FONT_5X12:ARRAY[0..255,0..9]OF BYTE :=[
16#00,16#00,16#00,16#00,16#00,16#00,16#00,16#00,16#00,16#00,	// 16#00
16#FE,16#01,16#49,16#02,16#81,16#02,16#49,16#02,16#FE,16#01,	// 16#01
16#FE,16#01,16#B7,16#03,16#7F,16#03,16#B7,16#03,16#FE,16#01,	// 16#02
16#7C,16#00,16#FE,16#01,16#F8,16#07,16#FE,16#01,16#7C,16#00,	// 16#03
16#70,16#00,16#FC,16#01,16#FF,16#07,16#FC,16#01,16#70,16#00,	// 16#04
16#60,16#00,16#EE,16#02,16#FF,16#03,16#EE,16#02,16#60,16#00,	// 16#05
16#70,16#00,16#FC,16#02,16#FF,16#03,16#FC,16#02,16#70,16#00,	// 16#06
16#00,16#00,16#00,16#00,16#00,16#00,16#00,16#00,16#00,16#00,	// 16#07
16#00,16#00,16#00,16#00,16#00,16#00,16#00,16#00,16#00,16#00,	// 16#08
16#00,16#00,16#00,16#00,16#00,16#00,16#00,16#00,16#00,16#00,	// 16#09
16#00,16#00,16#00,16#00,16#00,16#00,16#00,16#00,16#00,16#00,	// 16#0A
16#C0,16#01,16#20,16#02,16#34,16#02,16#CC,16#01,16#1C,16#00,	// 16#0B
16#1C,16#01,16#E2,16#03,16#22,16#01,16#1C,16#00,16#00,16#00,	// 16#0C
16#00,16#00,16#00,16#00,16#00,16#00,16#00,16#00,16#00,16#00,	// 16#0D
16#00,16#03,16#FE,16#03,16#C5,16#00,16#FF,16#00,16#00,16#00,	// 16#0E
16#50,16#01,16#A0,16#00,16#B0,16#01,16#A0,16#00,16#50,16#01,	// 16#0F
16#FC,16#01,16#F8,16#00,16#70,16#00,16#20,16#00,16#00,16#00,	// 16#10
16#20,16#00,16#70,16#00,16#F8,16#00,16#FC,16#01,16#00,16#00,	// 16#11
16#88,16#00,16#04,16#01,16#FE,16#03,16#04,16#01,16#88,16#00,	// 16#12
16#00,16#00,16#7C,16#03,16#00,16#00,16#7C,16#03,16#00,16#00,	// 16#13
16#3C,16#00,16#FE,16#03,16#02,16#00,16#FE,16#03,16#00,16#00,	// 16#14
16#2C,16#01,16#52,16#02,16#52,16#02,16#A4,16#01,16#00,16#00,	// 16#15
16#00,16#03,16#00,16#03,16#00,16#03,16#00,16#03,16#00,16#00,	// 16#16
16#88,16#04,16#04,16#05,16#FE,16#07,16#04,16#05,16#88,16#04,	// 16#17
16#08,16#00,16#04,16#00,16#FE,16#03,16#04,16#00,16#08,16#00,	// 16#18
16#80,16#00,16#00,16#01,16#FC,16#03,16#00,16#01,16#80,16#00,	// 16#19
16#20,16#00,16#A8,16#00,16#70,16#00,16#20,16#00,16#00,16#00,	// 16#1A
16#20,16#00,16#70,16#00,16#A8,16#00,16#20,16#00,16#00,16#00,	// 16#1B
16#E0,16#00,16#80,16#00,16#80,16#00,16#80,16#00,16#00,16#00,	// 16#1C
16#20,16#00,16#F8,16#00,16#20,16#00,16#F8,16#00,16#20,16#00,	// 16#1D
16#80,16#00,16#E0,16#00,16#F8,16#00,16#E0,16#00,16#80,16#00,	// 16#1E
16#08,16#00,16#38,16#00,16#F8,16#00,16#38,16#00,16#08,16#00,	// 16#1F
16#00,16#00,16#00,16#00,16#00,16#00,16#00,16#00,16#00,16#00,	// 16#20
16#00,16#00,16#00,16#00,16#7E,16#03,16#00,16#00,16#00,16#00,	// 16#21
16#00,16#00,16#0F,16#00,16#00,16#00,16#0F,16#00,16#00,16#00,	// 16#22
16#48,16#00,16#FE,16#01,16#48,16#00,16#FE,16#01,16#48,16#00,	// 16#23
16#18,16#01,16#26,16#02,16#44,16#06,16#88,16#01,16#00,16#00,	// 16#24
16#06,16#03,16#E6,16#00,16#18,16#03,16#06,16#03,16#00,16#00,	// 16#25
16#DC,16#01,16#22,16#02,16#5C,16#02,16#80,16#01,16#40,16#02,	// 16#26
16#00,16#00,16#00,16#00,16#0B,16#00,16#07,16#00,16#00,16#00,	// 16#27
16#00,16#00,16#FC,16#01,16#02,16#02,16#00,16#00,16#00,16#00,	// 16#28
16#00,16#00,16#02,16#02,16#FC,16#01,16#00,16#00,16#00,16#00,	// 16#29
16#48,16#00,16#30,16#00,16#FC,16#00,16#30,16#00,16#48,16#00,	// 16#2A
16#20,16#00,16#20,16#00,16#F8,16#00,16#20,16#00,16#20,16#00,	// 16#2B
16#00,16#00,16#00,16#0B,16#00,16#07,16#00,16#00,16#00,16#00,	// 16#2C
16#20,16#00,16#20,16#00,16#20,16#00,16#20,16#00,16#00,16#00,	// 16#2D
16#00,16#00,16#00,16#03,16#00,16#03,16#00,16#00,16#00,16#00,	// 16#2E
16#00,16#03,16#E0,16#00,16#18,16#00,16#06,16#00,16#00,16#00,	// 16#2F
16#FC,16#03,16#02,16#02,16#02,16#02,16#FE,16#01,16#00,16#00,	// 16#30
16#08,16#02,16#04,16#02,16#FE,16#03,16#00,16#02,16#00,16#00,	// 16#31
16#8C,16#03,16#42,16#02,16#22,16#02,16#1C,16#02,16#00,16#00,	// 16#32
16#04,16#01,16#22,16#02,16#22,16#02,16#DC,16#01,16#00,16#00,	// 16#33
16#60,16#00,16#58,16#00,16#44,16#00,16#FE,16#03,16#00,16#00,	// 16#34
16#3E,16#01,16#22,16#02,16#22,16#02,16#C2,16#01,16#00,16#00,	// 16#35
16#F8,16#01,16#14,16#02,16#12,16#02,16#E2,16#01,16#00,16#00,	// 16#36
16#02,16#00,16#82,16#03,16#62,16#00,16#1E,16#00,16#00,16#00,	// 16#37
16#DC,16#01,16#22,16#02,16#22,16#02,16#DC,16#01,16#00,16#00,	// 16#38
16#3C,16#02,16#42,16#02,16#42,16#01,16#FC,16#00,16#00,16#00,	// 16#39
16#00,16#00,16#30,16#03,16#30,16#03,16#00,16#00,16#00,16#00,	// 16#3A
16#00,16#00,16#30,16#0B,16#30,16#07,16#00,16#00,16#00,16#00,	// 16#3B
16#60,16#00,16#90,16#00,16#08,16#01,16#04,16#02,16#00,16#00,	// 16#3C
16#A0,16#00,16#A0,16#00,16#A0,16#00,16#A0,16#00,16#00,16#00,	// 16#3D
16#04,16#02,16#08,16#01,16#90,16#00,16#60,16#00,16#00,16#00,	// 16#3E
16#0C,16#00,16#02,16#00,16#62,16#03,16#1C,16#00,16#00,16#00,	// 16#3F
16#FC,16#01,16#02,16#02,16#62,16#02,16#7C,16#02,16#00,16#00,	// 16#40
16#FC,16#03,16#22,16#00,16#22,16#00,16#FC,16#03,16#00,16#00,	// 16#41
16#FE,16#03,16#22,16#02,16#22,16#02,16#DC,16#01,16#00,16#00,	// 16#42
16#FC,16#01,16#02,16#02,16#02,16#02,16#0C,16#01,16#00,16#00,	// 16#43
16#FE,16#03,16#02,16#02,16#02,16#02,16#FC,16#01,16#00,16#00,	// 16#44
16#FE,16#03,16#22,16#02,16#22,16#02,16#22,16#02,16#00,16#00,	// 16#45
16#FE,16#03,16#22,16#00,16#22,16#00,16#22,16#00,16#00,16#00,	// 16#46
16#FC,16#01,16#02,16#02,16#42,16#02,16#CC,16#01,16#00,16#00,	// 16#47
16#FE,16#03,16#20,16#00,16#20,16#00,16#FE,16#03,16#00,16#00,	// 16#48
16#00,16#00,16#02,16#02,16#FE,16#03,16#02,16#02,16#00,16#00,	// 16#49
16#80,16#01,16#02,16#02,16#FE,16#01,16#02,16#00,16#00,16#00,	// 16#4A
16#FE,16#03,16#20,16#00,16#D8,16#00,16#06,16#03,16#00,16#00,	// 16#4B
16#FE,16#03,16#00,16#02,16#00,16#02,16#00,16#02,16#00,16#00,	// 16#4C
16#FE,16#03,16#18,16#00,16#18,16#00,16#FE,16#03,16#00,16#00,	// 16#4D
16#FE,16#03,16#18,16#00,16#60,16#00,16#FE,16#03,16#00,16#00,	// 16#4E
16#FC,16#01,16#02,16#02,16#02,16#02,16#FC,16#01,16#00,16#00,	// 16#4F
16#FE,16#03,16#22,16#00,16#22,16#00,16#1C,16#00,16#00,16#00,	// 16#50
16#FC,16#01,16#02,16#02,16#02,16#06,16#FC,16#09,16#00,16#00,	// 16#51
16#FE,16#03,16#62,16#00,16#A2,16#00,16#1C,16#03,16#00,16#00,	// 16#52
16#9C,16#01,16#22,16#02,16#22,16#02,16#CC,16#01,16#00,16#00,	// 16#53
16#02,16#00,16#02,16#00,16#FE,16#03,16#02,16#00,16#02,16#00,	// 16#54
16#FE,16#01,16#00,16#02,16#00,16#02,16#FE,16#01,16#00,16#00,	// 16#55
16#3E,16#00,16#C0,16#00,16#00,16#03,16#FE,16#00,16#00,16#00,	// 16#56
16#FE,16#03,16#80,16#00,16#80,16#00,16#FE,16#03,16#00,16#00,	// 16#57
16#8E,16#03,16#70,16#00,16#70,16#00,16#8E,16#03,16#00,16#00,	// 16#58
16#0E,16#00,16#30,16#00,16#C0,16#03,16#30,16#00,16#0E,16#00,	// 16#59
16#82,16#03,16#62,16#02,16#1A,16#02,16#06,16#02,16#00,16#00,	// 16#5A
16#00,16#00,16#FE,16#03,16#02,16#02,16#00,16#00,16#00,16#00,	// 16#5B
16#06,16#00,16#18,16#00,16#E0,16#00,16#00,16#03,16#00,16#00,	// 16#5C
16#00,16#00,16#02,16#02,16#FE,16#03,16#00,16#00,16#00,16#00,	// 16#5D
16#00,16#00,16#04,16#00,16#02,16#00,16#04,16#00,16#00,16#00,	// 16#5E
16#00,16#08,16#00,16#08,16#00,16#08,16#00,16#08,16#00,16#08,	// 16#5F
16#00,16#00,16#07,16#00,16#0B,16#00,16#00,16#00,16#00,16#00,	// 16#60
16#80,16#01,16#50,16#02,16#50,16#02,16#E0,16#03,16#00,16#00,	// 16#61
16#FE,16#03,16#10,16#02,16#10,16#02,16#E0,16#01,16#00,16#00,	// 16#62
16#E0,16#01,16#10,16#02,16#10,16#02,16#10,16#02,16#00,16#00,	// 16#63
16#E0,16#01,16#10,16#02,16#10,16#02,16#FE,16#03,16#00,16#00,	// 16#64
16#E0,16#01,16#90,16#02,16#90,16#02,16#E0,16#02,16#00,16#00,	// 16#65
16#10,16#00,16#FC,16#03,16#12,16#00,16#00,16#00,16#00,16#00,	// 16#66
16#E0,16#01,16#10,16#0A,16#10,16#0A,16#F0,16#07,16#00,16#00,	// 16#67
16#FE,16#03,16#10,16#00,16#10,16#00,16#E0,16#03,16#00,16#00,	// 16#68
16#00,16#00,16#00,16#02,16#F4,16#03,16#00,16#02,16#00,16#00,	// 16#69
16#00,16#04,16#00,16#08,16#F4,16#07,16#00,16#00,16#00,16#00,	// 16#6A
16#FE,16#03,16#C0,16#00,16#20,16#01,16#10,16#02,16#00,16#00,	// 16#6B
16#00,16#00,16#02,16#02,16#FE,16#03,16#00,16#02,16#00,16#00,	// 16#6C
16#F0,16#03,16#20,16#00,16#20,16#00,16#F0,16#03,16#00,16#00,	// 16#6D
16#F0,16#03,16#20,16#00,16#10,16#00,16#E0,16#03,16#00,16#00,	// 16#6E
16#E0,16#01,16#10,16#02,16#10,16#02,16#E0,16#01,16#00,16#00,	// 16#6F
16#F0,16#0F,16#10,16#02,16#10,16#02,16#E0,16#01,16#00,16#00,	// 16#70
16#E0,16#01,16#10,16#02,16#10,16#02,16#F0,16#0F,16#00,16#00,	// 16#71
16#10,16#00,16#E0,16#03,16#10,16#00,16#30,16#00,16#00,16#00,	// 16#72
16#20,16#01,16#50,16#02,16#90,16#02,16#20,16#01,16#00,16#00,	// 16#73
16#10,16#00,16#FC,16#03,16#10,16#02,16#00,16#00,16#00,16#00,	// 16#74
16#F0,16#01,16#00,16#02,16#00,16#02,16#F0,16#03,16#00,16#00,	// 16#75
16#30,16#00,16#C0,16#00,16#00,16#03,16#F0,16#00,16#00,16#00,	// 16#76
16#F0,16#03,16#00,16#01,16#00,16#01,16#F0,16#03,16#00,16#00,	// 16#77
16#30,16#03,16#C0,16#00,16#C0,16#00,16#30,16#03,16#00,16#00,	// 16#78
16#F0,16#09,16#00,16#0A,16#00,16#0A,16#F0,16#07,16#00,16#00,	// 16#79
16#10,16#03,16#90,16#02,16#50,16#02,16#30,16#02,16#00,16#00,	// 16#7A
16#20,16#00,16#DC,16#01,16#02,16#02,16#00,16#00,16#00,16#00,	// 16#7B
16#00,16#00,16#00,16#00,16#EF,16#03,16#00,16#00,16#00,16#00,	// 16#7C
16#00,16#00,16#02,16#02,16#DC,16#01,16#20,16#00,16#00,16#00,	// 16#7D
16#04,16#00,16#02,16#00,16#04,16#00,16#02,16#00,16#00,16#00,	// 16#7E
16#E0,16#03,16#18,16#02,16#06,16#02,16#18,16#02,16#E0,16#03,	// 16#7F
16#FC,16#01,16#02,16#0A,16#02,16#06,16#0C,16#01,16#00,16#00,	// 16#80
16#F0,16#01,16#06,16#02,16#00,16#02,16#F6,16#03,16#00,16#00,	// 16#81
16#E0,16#01,16#94,16#02,16#92,16#02,16#E2,16#02,16#00,16#00,	// 16#82
16#24,16#01,16#92,16#02,16#92,16#02,16#E4,16#03,16#00,16#00,	// 16#83
16#20,16#01,16#96,16#02,16#90,16#02,16#E6,16#03,16#00,16#00,	// 16#84
16#22,16#01,16#92,16#02,16#94,16#02,16#E0,16#03,16#00,16#00,	// 16#85
16#20,16#01,16#94,16#02,16#9A,16#02,16#E4,16#03,16#00,16#00,	// 16#86
16#E0,16#09,16#10,16#0A,16#10,16#06,16#10,16#02,16#00,16#00,	// 16#87
16#E4,16#01,16#92,16#02,16#92,16#02,16#E4,16#02,16#00,16#00,	// 16#88
16#E0,16#01,16#96,16#02,16#90,16#02,16#E6,16#02,16#00,16#00,	// 16#89
16#E2,16#01,16#92,16#02,16#94,16#02,16#E0,16#02,16#00,16#00,	// 16#8A
16#00,16#00,16#16,16#02,16#F0,16#03,16#06,16#02,16#00,16#00,	// 16#8B
16#04,16#00,16#12,16#02,16#F2,16#03,16#04,16#02,16#00,16#00,	// 16#8C
16#00,16#00,16#12,16#02,16#F2,16#03,16#04,16#02,16#00,16#00,	// 16#8D
16#F8,16#03,16#45,16#00,16#44,16#00,16#F9,16#03,16#00,16#00,	// 16#8E
16#F0,16#03,16#4A,16#00,16#4D,16#00,16#F2,16#03,16#00,16#00,	// 16#8F
16#F8,16#03,16#4A,16#02,16#49,16#02,16#49,16#02,16#00,16#00,	// 16#90
16#00,16#01,16#90,16#02,16#F0,16#01,16#90,16#02,16#60,16#00,	// 16#91
16#F8,16#03,16#4C,16#00,16#FC,16#03,16#44,16#02,16#00,16#00,	// 16#92
16#E4,16#01,16#12,16#02,16#12,16#02,16#E4,16#01,16#00,16#00,	// 16#93
16#E0,16#01,16#16,16#02,16#10,16#02,16#E6,16#01,16#00,16#00,	// 16#94
16#E0,16#01,16#12,16#02,16#12,16#02,16#E4,16#01,16#00,16#00,	// 16#95
16#F4,16#01,16#02,16#02,16#02,16#02,16#F4,16#03,16#00,16#00,	// 16#96
16#F2,16#01,16#02,16#02,16#04,16#02,16#F0,16#03,16#00,16#00,	// 16#97
16#F0,16#09,16#06,16#0A,16#00,16#0A,16#F6,16#07,16#00,16#00,	// 16#98
16#F8,16#01,16#05,16#02,16#04,16#02,16#F9,16#01,16#00,16#00,	// 16#99
16#FC,16#01,16#01,16#02,16#00,16#02,16#FD,16#03,16#00,16#00,	// 16#9A
16#E0,16#03,16#90,16#01,16#70,16#01,16#F8,16#00,16#00,16#00,	// 16#9B
16#20,16#03,16#FC,16#03,16#22,16#02,16#04,16#03,16#00,16#00,	// 16#9C
16#FE,16#03,16#E1,16#03,16#1D,16#02,16#FF,16#01,16#00,16#00,	// 16#9D
16#88,16#00,16#50,16#00,16#20,16#00,16#50,16#00,16#88,16#00,	// 16#9E
16#00,16#04,16#20,16#08,16#FE,16#07,16#21,16#00,16#00,16#00,	// 16#9F
16#20,16#01,16#94,16#02,16#92,16#02,16#E2,16#03,16#00,16#00,	// 16#A0
16#00,16#00,16#14,16#02,16#F2,16#03,16#02,16#02,16#00,16#00,	// 16#A1
16#E0,16#01,16#14,16#02,16#12,16#02,16#E2,16#01,16#00,16#00,	// 16#A2
16#F0,16#01,16#04,16#02,16#02,16#02,16#F2,16#03,16#00,16#00,	// 16#A3
16#F4,16#03,16#22,16#00,16#14,16#00,16#E2,16#03,16#00,16#00,	// 16#A4
16#FA,16#03,16#31,16#00,16#62,16#00,16#F9,16#03,16#00,16#00,	// 16#A5
16#90,16#00,16#AA,16#00,16#AA,16#00,16#BC,16#00,16#00,16#00,	// 16#A6
16#9C,16#00,16#A2,16#00,16#A2,16#00,16#9C,16#00,16#00,16#00,	// 16#A7
16#C0,16#01,16#36,16#02,16#00,16#02,16#00,16#01,16#00,16#00,	// 16#A8
16#F8,16#01,16#F4,16#02,16#54,16#02,16#A4,16#02,16#F8,16#01,	// 16#A9
16#40,16#00,16#40,16#00,16#40,16#00,16#C0,16#01,16#00,16#00,	// 16#AA
16#80,16#01,16#6E,16#00,16#50,16#03,16#CC,16#02,16#00,16#00,	// 16#AB
16#80,16#01,16#6E,16#00,16#90,16#01,16#CC,16#03,16#00,16#00,	// 16#AC
16#00,16#00,16#00,16#00,16#F4,16#03,16#00,16#00,16#00,16#00,	// 16#AD
16#60,16#00,16#98,16#01,16#60,16#00,16#98,16#01,16#00,16#00,	// 16#AE
16#98,16#01,16#60,16#00,16#98,16#01,16#60,16#00,16#00,16#00,	// 16#AF
16#04,16#01,16#20,16#08,16#04,16#01,16#20,16#08,16#04,16#01,	// 16#B0
16#88,16#08,16#22,16#02,16#88,16#08,16#22,16#02,16#88,16#08,	// 16#B1
16#AA,16#0A,16#55,16#05,16#AA,16#0A,16#55,16#05,16#AA,16#0A,	// 16#B2
16#00,16#00,16#00,16#00,16#FF,16#0F,16#00,16#00,16#00,16#00,	// 16#B3
16#20,16#00,16#20,16#00,16#FF,16#0F,16#00,16#00,16#00,16#00,	// 16#B4
16#F0,16#03,16#4A,16#00,16#49,16#00,16#F1,16#03,16#00,16#00,	// 16#B5
16#F0,16#03,16#4A,16#00,16#49,16#00,16#F2,16#03,16#00,16#00,	// 16#B6
16#F1,16#03,16#49,16#00,16#4A,16#00,16#F0,16#03,16#00,16#00,	// 16#B7
16#F8,16#01,16#64,16#02,16#94,16#02,16#04,16#02,16#F8,16#01,	// 16#B8
16#50,16#00,16#DF,16#0F,16#00,16#00,16#FF,16#0F,16#00,16#00,	// 16#B9
16#00,16#00,16#FF,16#0F,16#00,16#00,16#FF,16#0F,16#00,16#00,	// 16#BA
16#50,16#00,16#D0,16#0F,16#10,16#00,16#F0,16#0F,16#00,16#00,	// 16#BB
16#50,16#00,16#5F,16#00,16#40,16#00,16#7F,16#00,16#00,16#00,	// 16#BC
16#E0,16#00,16#10,16#01,16#18,16#03,16#10,16#01,16#A0,16#00,	// 16#BD
16#52,16#00,16#5C,16#00,16#F0,16#03,16#5C,16#00,16#52,16#00,	// 16#BE
16#20,16#00,16#20,16#00,16#E0,16#0F,16#00,16#00,16#00,16#00,	// 16#BF
16#00,16#00,16#00,16#00,16#3F,16#00,16#20,16#00,16#20,16#00,	// 16#C0
16#20,16#00,16#20,16#00,16#3F,16#00,16#20,16#00,16#20,16#00,	// 16#C1
16#20,16#00,16#20,16#00,16#E0,16#0F,16#20,16#00,16#20,16#00,	// 16#C2
16#00,16#00,16#00,16#00,16#FF,16#0F,16#20,16#00,16#20,16#00,	// 16#C3
16#20,16#00,16#20,16#00,16#20,16#00,16#20,16#00,16#20,16#00,	// 16#C4
16#20,16#00,16#20,16#00,16#FF,16#0F,16#20,16#00,16#20,16#00,	// 16#C5
16#24,16#01,16#92,16#02,16#94,16#02,16#E2,16#03,16#00,16#00,	// 16#C6
16#F2,16#03,16#49,16#00,16#4A,16#00,16#F1,16#03,16#00,16#00,	// 16#C7
16#00,16#00,16#7F,16#00,16#40,16#00,16#5F,16#00,16#50,16#00,	// 16#C8
16#00,16#00,16#F0,16#0F,16#10,16#00,16#D0,16#0F,16#50,16#00,	// 16#C9
16#50,16#00,16#5F,16#00,16#40,16#00,16#5F,16#00,16#50,16#00,	// 16#CA
16#50,16#00,16#D0,16#0F,16#10,16#00,16#D0,16#0F,16#50,16#00,	// 16#CB
16#00,16#00,16#FF,16#0F,16#00,16#00,16#DF,16#0F,16#50,16#00,	// 16#CC
16#50,16#00,16#50,16#00,16#50,16#00,16#50,16#00,16#50,16#00,	// 16#CD
16#50,16#00,16#DF,16#0F,16#00,16#00,16#DF,16#0F,16#50,16#00,	// 16#CE
16#FA,16#02,16#04,16#01,16#04,16#01,16#FA,16#02,16#00,16#00,	// 16#CF
16#80,16#01,16#58,16#02,16#64,16#02,16#C4,16#01,16#00,16#00,	// 16#D0
16#20,16#00,16#FE,16#03,16#22,16#02,16#FC,16#01,16#00,16#00,	// 16#D1
16#F8,16#03,16#4A,16#02,16#49,16#02,16#4A,16#02,16#00,16#00,	// 16#D2
16#F8,16#03,16#4A,16#02,16#48,16#02,16#4A,16#02,16#00,16#00,	// 16#D3
16#F8,16#03,16#49,16#02,16#49,16#02,16#4A,16#02,16#00,16#00,	// 16#D4
16#00,16#00,16#00,16#00,16#1E,16#00,16#00,16#00,16#00,16#00,	// 16#D5
16#00,16#00,16#0A,16#02,16#F9,16#03,16#09,16#02,16#00,16#00,	// 16#D6
16#00,16#00,16#0A,16#02,16#F9,16#03,16#0A,16#02,16#00,16#00,	// 16#D7
16#00,16#00,16#0A,16#02,16#F8,16#03,16#0A,16#02,16#00,16#00,	// 16#D8
16#20,16#00,16#20,16#00,16#3F,16#00,16#00,16#00,16#00,16#00,	// 16#D9
16#00,16#00,16#00,16#00,16#E0,16#0F,16#20,16#00,16#20,16#00,	// 16#DA
16#FF,16#0F,16#FF,16#0F,16#FF,16#0F,16#FF,16#0F,16#FF,16#0F,	// 16#DB
16#C0,16#0F,16#C0,16#0F,16#C0,16#0F,16#C0,16#0F,16#C0,16#0F,	// 16#DC
16#00,16#00,16#00,16#00,16#EF,16#03,16#00,16#00,16#00,16#00,	// 16#DD
16#00,16#00,16#09,16#02,16#F9,16#03,16#0A,16#02,16#00,16#00,	// 16#DE
16#3F,16#00,16#3F,16#00,16#3F,16#00,16#3F,16#00,16#3F,16#00,	// 16#DF
16#F0,16#01,16#0A,16#02,16#09,16#02,16#F1,16#01,16#00,16#00,	// 16#E0
16#FC,16#0F,16#22,16#02,16#32,16#02,16#CC,16#01,16#00,16#00,	// 16#E1
16#F0,16#01,16#0A,16#02,16#09,16#02,16#F2,16#01,16#00,16#00,	// 16#E2
16#F0,16#01,16#09,16#02,16#09,16#02,16#F2,16#01,16#00,16#00,	// 16#E3
16#E4,16#01,16#12,16#02,16#14,16#02,16#E2,16#01,16#00,16#00,	// 16#E4
16#F2,16#01,16#09,16#02,16#0A,16#02,16#F1,16#01,16#00,16#00,	// 16#E5
16#F0,16#0F,16#00,16#02,16#00,16#02,16#F0,16#01,16#00,16#00,	// 16#E6
16#F8,16#03,16#A8,16#02,16#A0,16#00,16#40,16#00,16#00,16#00,	// 16#E7
16#FE,16#03,16#8A,16#02,16#88,16#00,16#70,16#00,16#00,16#00,	// 16#E8
16#F8,16#01,16#02,16#02,16#01,16#02,16#F9,16#01,16#00,16#00,	// 16#E9
16#F8,16#01,16#02,16#02,16#01,16#02,16#FA,16#01,16#00,16#00,	// 16#EA
16#F8,16#01,16#01,16#02,16#01,16#02,16#FA,16#01,16#00,16#00,	// 16#EB
16#F0,16#09,16#04,16#0A,16#02,16#0A,16#F2,16#07,16#00,16#00,	// 16#EC
16#18,16#00,16#62,16#00,16#81,16#03,16#61,16#00,16#18,16#00,	// 16#ED
16#00,16#00,16#04,16#00,16#04,16#00,16#04,16#00,16#00,16#00,	// 16#EE
16#00,16#00,16#0B,16#00,16#07,16#00,16#00,16#00,16#00,16#00,	// 16#EF
16#20,16#00,16#20,16#00,16#20,16#00,16#20,16#00,16#00,16#00,	// 16#F0
16#20,16#02,16#20,16#02,16#F8,16#02,16#20,16#02,16#20,16#02,	// 16#F1
16#A0,16#00,16#A0,16#00,16#A0,16#00,16#A0,16#00,16#00,16#00,	// 16#F2
16#89,16#01,16#6B,16#00,16#95,16#01,16#CC,16#03,16#00,16#00,	// 16#F3
16#3C,16#00,16#FE,16#03,16#02,16#00,16#FE,16#03,16#00,16#00,	// 16#F4
16#2C,16#01,16#52,16#02,16#52,16#02,16#A4,16#01,16#00,16#00,	// 16#F5
16#20,16#00,16#20,16#00,16#A8,16#00,16#20,16#00,16#20,16#00,	// 16#F6
16#20,16#00,16#40,16#00,16#60,16#00,16#60,16#00,16#00,16#00,	// 16#F7
16#06,16#00,16#09,16#00,16#09,16#00,16#06,16#00,16#00,16#00,	// 16#F8
16#00,16#00,16#60,16#00,16#00,16#00,16#60,16#00,16#00,16#00,	// 16#F9
16#00,16#00,16#00,16#00,16#60,16#00,16#00,16#00,16#00,16#00,	// 16#FA
16#00,16#00,16#02,16#00,16#3F,16#00,16#00,16#00,16#00,16#00,	// 16#FB
16#11,16#00,16#25,16#00,16#25,16#00,16#1B,16#00,16#00,16#00,	// 16#FC
16#32,16#00,16#29,16#00,16#29,16#00,16#26,16#00,16#00,16#00,	// 16#FD
16#00,16#00,16#F8,16#00,16#F8,16#00,16#F8,16#00,16#00,16#00,	// 16#FE
16#00,16#00,16#00,16#00,16#00,16#00,16#00,16#00,16#00,16#00 	// 16#FF
];


FONT_6X8:ARRAY[0..255,0..5]OF BYTE :=[
16#00,16#00,16#00,16#00,16#00,16#00,	// 16#00
16#00,16#3E,16#45,16#51,16#45,16#3E,	// 16#01
16#00,16#3E,16#6B,16#6F,16#6B,16#3E,	// 16#02
16#00,16#1C,16#3E,16#7C,16#3E,16#1C,	// 16#03
16#00,16#18,16#3C,16#7E,16#3C,16#18,	// 16#04
16#00,16#30,16#36,16#7F,16#36,16#30,	// 16#05
16#00,16#18,16#5C,16#7E,16#5C,16#18,	// 16#06
16#00,16#00,16#00,16#00,16#00,16#00,	// 16#07
16#00,16#00,16#00,16#00,16#00,16#00,	// 16#08
16#00,16#00,16#00,16#00,16#00,16#00,	// 16#09
16#00,16#00,16#00,16#00,16#00,16#00,	// 16#0A
16#00,16#30,16#48,16#4A,16#36,16#0E,	// 16#0B
16#00,16#06,16#29,16#79,16#29,16#06,	// 16#0C
16#00,16#00,16#00,16#00,16#00,16#00,	// 16#0D
16#00,16#60,16#7E,16#0A,16#35,16#3F,	// 16#0E
16#00,16#2A,16#1C,16#36,16#1C,16#2A,	// 16#0F
16#00,16#00,16#7F,16#3E,16#1C,16#08,	// 16#10
16#00,16#08,16#1C,16#3E,16#7F,16#00,	// 16#11
16#00,16#14,16#36,16#7F,16#36,16#14,	// 16#12
16#00,16#00,16#5F,16#00,16#5F,16#00,	// 16#13
16#00,16#06,16#09,16#7F,16#01,16#7F,	// 16#14
16#00,16#22,16#4D,16#55,16#59,16#22,	// 16#15
16#00,16#60,16#60,16#60,16#60,16#00,	// 16#16
16#00,16#14,16#B6,16#FF,16#B6,16#14,	// 16#17
16#00,16#04,16#06,16#7F,16#06,16#04,	// 16#18
16#00,16#10,16#30,16#7F,16#30,16#10,	// 16#19
16#00,16#08,16#08,16#3E,16#1C,16#08,	// 16#1A
16#00,16#08,16#1C,16#3E,16#08,16#08,	// 16#1B
16#00,16#78,16#40,16#40,16#40,16#40,	// 16#1C
16#00,16#08,16#3E,16#08,16#3E,16#08,	// 16#1D
16#00,16#30,16#3C,16#3F,16#3C,16#30,	// 16#1E
16#00,16#03,16#0F,16#3F,16#0F,16#03,	// 16#1F
16#00,16#00,16#00,16#00,16#00,16#00,	// 16#20
16#00,16#00,16#06,16#5F,16#06,16#00,	// 16#21
16#00,16#07,16#03,16#00,16#07,16#03,	// 16#22
16#00,16#24,16#7E,16#24,16#7E,16#24,	// 16#23
16#00,16#24,16#2B,16#6A,16#12,16#00,	// 16#24
16#00,16#63,16#13,16#08,16#64,16#63,	// 16#25
16#00,16#36,16#49,16#56,16#20,16#50,	// 16#26
16#00,16#00,16#07,16#03,16#00,16#00,	// 16#27
16#00,16#00,16#3E,16#41,16#00,16#00,	// 16#28
16#00,16#00,16#41,16#3E,16#00,16#00,	// 16#29
16#00,16#08,16#3E,16#1C,16#3E,16#08,	// 16#2A
16#00,16#08,16#08,16#3E,16#08,16#08,	// 16#2B
16#00,16#00,16#E0,16#60,16#00,16#00,	// 16#2C
16#00,16#08,16#08,16#08,16#08,16#08,	// 16#2D
16#00,16#00,16#60,16#60,16#00,16#00,	// 16#2E
16#00,16#20,16#10,16#08,16#04,16#02,	// 16#2F
16#00,16#3E,16#51,16#49,16#45,16#3E,	// 16#30
16#00,16#00,16#42,16#7F,16#40,16#00,	// 16#31
16#00,16#62,16#51,16#49,16#49,16#46,	// 16#32
16#00,16#22,16#49,16#49,16#49,16#36,	// 16#33
16#00,16#18,16#14,16#12,16#7F,16#10,	// 16#34
16#00,16#2F,16#49,16#49,16#49,16#31,	// 16#35
16#00,16#3C,16#4A,16#49,16#49,16#30,	// 16#36
16#00,16#01,16#71,16#09,16#05,16#03,	// 16#37
16#00,16#36,16#49,16#49,16#49,16#36,	// 16#38
16#00,16#06,16#49,16#49,16#29,16#1E,	// 16#39
16#00,16#00,16#6C,16#6C,16#00,16#00,	// 16#3A
16#00,16#00,16#EC,16#6C,16#00,16#00,	// 16#3B
16#00,16#08,16#14,16#22,16#41,16#00,	// 16#3C
16#00,16#24,16#24,16#24,16#24,16#24,	// 16#3D
16#00,16#00,16#41,16#22,16#14,16#08,	// 16#3E
16#00,16#02,16#01,16#59,16#09,16#06,	// 16#3F
16#00,16#3E,16#41,16#5D,16#55,16#1E,	// 16#40
16#00,16#7E,16#11,16#11,16#11,16#7E,	// 16#41
16#00,16#7F,16#49,16#49,16#49,16#36,	// 16#42
16#00,16#3E,16#41,16#41,16#41,16#22,	// 16#43
16#00,16#7F,16#41,16#41,16#41,16#3E,	// 16#44
16#00,16#7F,16#49,16#49,16#49,16#41,	// 16#45
16#00,16#7F,16#09,16#09,16#09,16#01,	// 16#46
16#00,16#3E,16#41,16#49,16#49,16#7A,	// 16#47
16#00,16#7F,16#08,16#08,16#08,16#7F,	// 16#48
16#00,16#00,16#41,16#7F,16#41,16#00,	// 16#49
16#00,16#30,16#40,16#40,16#40,16#3F,	// 16#4A
16#00,16#7F,16#08,16#14,16#22,16#41,	// 16#4B
16#00,16#7F,16#40,16#40,16#40,16#40,	// 16#4C
16#00,16#7F,16#02,16#04,16#02,16#7F,	// 16#4D
16#00,16#7F,16#02,16#04,16#08,16#7F,	// 16#4E
16#00,16#3E,16#41,16#41,16#41,16#3E,	// 16#4F
16#00,16#7F,16#09,16#09,16#09,16#06,	// 16#50
16#00,16#3E,16#41,16#51,16#21,16#5E,	// 16#51
16#00,16#7F,16#09,16#09,16#19,16#66,	// 16#52
16#00,16#26,16#49,16#49,16#49,16#32,	// 16#53
16#00,16#01,16#01,16#7F,16#01,16#01,	// 16#54
16#00,16#3F,16#40,16#40,16#40,16#3F,	// 16#55
16#00,16#1F,16#20,16#40,16#20,16#1F,	// 16#56
16#00,16#3F,16#40,16#3C,16#40,16#3F,	// 16#57
16#00,16#63,16#14,16#08,16#14,16#63,	// 16#58
16#00,16#07,16#08,16#70,16#08,16#07,	// 16#59
16#00,16#71,16#49,16#45,16#43,16#00,	// 16#5A
16#00,16#00,16#7F,16#41,16#41,16#00,	// 16#5B
16#00,16#02,16#04,16#08,16#10,16#20,	// 16#5C
16#00,16#00,16#41,16#41,16#7F,16#00,	// 16#5D
16#00,16#04,16#02,16#01,16#02,16#04,	// 16#5E
16#80,16#80,16#80,16#80,16#80,16#80,	// 16#5F
16#00,16#00,16#03,16#07,16#00,16#00,	// 16#60
16#00,16#20,16#54,16#54,16#54,16#78,	// 16#61
16#00,16#7F,16#44,16#44,16#44,16#38,	// 16#62
16#00,16#38,16#44,16#44,16#44,16#28,	// 16#63
16#00,16#38,16#44,16#44,16#44,16#7F,	// 16#64
16#00,16#38,16#54,16#54,16#54,16#08,	// 16#65
16#00,16#08,16#7E,16#09,16#09,16#00,	// 16#66
16#00,16#18,16#A4,16#A4,16#A4,16#7C,	// 16#67
16#00,16#7F,16#04,16#04,16#78,16#00,	// 16#68
16#00,16#00,16#00,16#7D,16#40,16#00,	// 16#69
16#00,16#40,16#80,16#84,16#7D,16#00,	// 16#6A
16#00,16#7F,16#10,16#28,16#44,16#00,	// 16#6B
16#00,16#00,16#00,16#7F,16#40,16#00,	// 16#6C
16#00,16#7C,16#04,16#18,16#04,16#78,	// 16#6D
16#00,16#7C,16#04,16#04,16#78,16#00,	// 16#6E
16#00,16#38,16#44,16#44,16#44,16#38,	// 16#6F
16#00,16#FC,16#44,16#44,16#44,16#38,	// 16#70
16#00,16#38,16#44,16#44,16#44,16#FC,	// 16#71
16#00,16#44,16#78,16#44,16#04,16#08,	// 16#72
16#00,16#08,16#54,16#54,16#54,16#20,	// 16#73
16#00,16#04,16#3E,16#44,16#24,16#00,	// 16#74
16#00,16#3C,16#40,16#20,16#7C,16#00,	// 16#75
16#00,16#1C,16#20,16#40,16#20,16#1C,	// 16#76
16#00,16#3C,16#60,16#30,16#60,16#3C,	// 16#77
16#00,16#6C,16#10,16#10,16#6C,16#00,	// 16#78
16#00,16#9C,16#A0,16#60,16#3C,16#00,	// 16#79
16#00,16#64,16#54,16#54,16#4C,16#00,	// 16#7A
16#00,16#08,16#3E,16#41,16#41,16#00,	// 16#7B
16#00,16#00,16#00,16#77,16#00,16#00,	// 16#7C
16#00,16#00,16#41,16#41,16#3E,16#08,	// 16#7D
16#00,16#02,16#01,16#02,16#01,16#00,	// 16#7E
16#00,16#3C,16#26,16#23,16#26,16#3C,	// 16#7F
16#00,16#1E,16#A1,16#E1,16#21,16#12,	// 16#80
16#00,16#3D,16#40,16#20,16#7D,16#00,	// 16#81
16#00,16#38,16#54,16#54,16#55,16#09,	// 16#82
16#00,16#20,16#55,16#55,16#55,16#78,	// 16#83
16#00,16#20,16#55,16#54,16#55,16#78,	// 16#84
16#00,16#20,16#55,16#55,16#54,16#78,	// 16#85
16#00,16#20,16#57,16#55,16#57,16#78,	// 16#86
16#00,16#1C,16#A2,16#E2,16#22,16#14,	// 16#87
16#00,16#38,16#55,16#55,16#55,16#08,	// 16#88
16#00,16#38,16#55,16#54,16#55,16#08,	// 16#89
16#00,16#38,16#55,16#55,16#54,16#08,	// 16#8A
16#00,16#00,16#01,16#7C,16#41,16#00,	// 16#8B
16#00,16#00,16#01,16#7D,16#41,16#00,	// 16#8C
16#00,16#00,16#01,16#7C,16#40,16#00,	// 16#8D
16#00,16#70,16#29,16#24,16#29,16#70,	// 16#8E
16#00,16#78,16#2F,16#25,16#2F,16#78,	// 16#8F
16#00,16#7C,16#54,16#54,16#55,16#45,	// 16#90
16#00,16#34,16#54,16#7C,16#54,16#58,	// 16#91
16#00,16#7E,16#09,16#7F,16#49,16#49,	// 16#92
16#00,16#38,16#45,16#45,16#39,16#00,	// 16#93
16#00,16#38,16#45,16#44,16#39,16#00,	// 16#94
16#00,16#39,16#45,16#44,16#38,16#00,	// 16#95
16#00,16#3C,16#41,16#21,16#7D,16#00,	// 16#96
16#00,16#3D,16#41,16#20,16#7C,16#00,	// 16#97
16#00,16#9C,16#A1,16#60,16#3D,16#00,	// 16#98
16#00,16#3D,16#42,16#42,16#3D,16#00,	// 16#99
16#00,16#3C,16#41,16#40,16#3D,16#00,	// 16#9A
16#80,16#70,16#68,16#58,16#38,16#04,	// 16#9B
16#00,16#48,16#3E,16#49,16#49,16#62,	// 16#9C
16#00,16#7E,16#61,16#5D,16#43,16#3F,	// 16#9D
16#00,16#22,16#14,16#08,16#14,16#22,	// 16#9E
16#00,16#40,16#88,16#7E,16#09,16#02,	// 16#9F
16#00,16#20,16#54,16#55,16#55,16#78,	// 16#A0
16#00,16#00,16#00,16#7D,16#41,16#00,	// 16#A1
16#00,16#38,16#44,16#45,16#39,16#00,	// 16#A2
16#00,16#3C,16#40,16#21,16#7D,16#00,	// 16#A3
16#00,16#7A,16#09,16#0A,16#71,16#00,	// 16#A4
16#00,16#7A,16#11,16#22,16#79,16#00,	// 16#A5
16#00,16#08,16#55,16#55,16#55,16#5E,	// 16#A6
16#00,16#4E,16#51,16#51,16#4E,16#00,	// 16#A7
16#00,16#30,16#48,16#4D,16#40,16#20,	// 16#A8
16#3E,16#41,16#5D,16#4B,16#55,16#3E,	// 16#A9
16#04,16#04,16#04,16#04,16#04,16#1C,	// 16#AA
16#00,16#17,16#08,16#4C,16#6A,16#50,	// 16#AB
16#00,16#17,16#08,16#34,16#2A,16#78,	// 16#AC
16#00,16#00,16#30,16#7D,16#30,16#00,	// 16#AD
16#00,16#08,16#14,16#00,16#08,16#14,	// 16#AE
16#00,16#14,16#08,16#00,16#14,16#08,	// 16#AF
16#44,16#11,16#44,16#11,16#44,16#11,	// 16#B0
16#AA,16#55,16#AA,16#55,16#AA,16#55,	// 16#B1
16#BB,16#EE,16#BB,16#EE,16#BB,16#EE,	// 16#B2
16#00,16#00,16#00,16#FF,16#00,16#00,	// 16#B3
16#08,16#08,16#08,16#FF,16#00,16#00,	// 16#B4
16#00,16#70,16#28,16#25,16#29,16#70,	// 16#B5
16#00,16#70,16#29,16#25,16#29,16#70,	// 16#B6
16#00,16#70,16#29,16#25,16#28,16#70,	// 16#B7
16#3E,16#41,16#5D,16#55,16#41,16#3E,	// 16#B8
16#0A,16#FB,16#00,16#FF,16#00,16#00,	// 16#B9
16#00,16#FF,16#00,16#FF,16#00,16#00,	// 16#BA
16#0A,16#FA,16#02,16#FE,16#00,16#00,	// 16#BB
16#0A,16#0B,16#08,16#0F,16#00,16#00,	// 16#BC
16#00,16#18,16#24,16#66,16#24,16#00,	// 16#BD
16#00,16#29,16#2A,16#7C,16#2A,16#29,	// 16#BE
16#08,16#08,16#08,16#F8,16#00,16#00,	// 16#BF
16#00,16#00,16#00,16#0F,16#08,16#08,	// 16#C0
16#08,16#08,16#08,16#0F,16#08,16#08,	// 16#C1
16#08,16#08,16#08,16#F8,16#08,16#08,	// 16#C2
16#00,16#00,16#00,16#FF,16#08,16#08,	// 16#C3
16#08,16#08,16#08,16#08,16#08,16#08,	// 16#C4
16#08,16#08,16#08,16#FF,16#08,16#08,	// 16#C5
16#00,16#20,16#56,16#55,16#56,16#79,	// 16#C6
16#00,16#70,16#2A,16#25,16#2A,16#71,	// 16#C7
16#00,16#0F,16#08,16#0B,16#0A,16#0A,	// 16#C8
16#00,16#FE,16#02,16#FA,16#0A,16#0A,	// 16#C9
16#0A,16#0B,16#08,16#0B,16#0A,16#0A,	// 16#CA
16#0A,16#FA,16#02,16#FA,16#0A,16#0A,	// 16#CB
16#00,16#FF,16#00,16#FB,16#0A,16#0A,	// 16#CC
16#0A,16#0A,16#0A,16#0A,16#0A,16#0A,	// 16#CD
16#0A,16#FB,16#00,16#FB,16#0A,16#0A,	// 16#CE
16#00,16#5D,16#22,16#22,16#22,16#5D,	// 16#CF
16#00,16#22,16#55,16#59,16#30,16#00,	// 16#D0
16#00,16#08,16#7F,16#49,16#41,16#3E,	// 16#D1
16#00,16#7C,16#55,16#55,16#55,16#44,	// 16#D2
16#00,16#7C,16#55,16#54,16#55,16#44,	// 16#D3
16#00,16#7C,16#55,16#55,16#54,16#44,	// 16#D4
16#00,16#00,16#00,16#07,16#00,16#00,	// 16#D5
16#00,16#00,16#44,16#7D,16#45,16#00,	// 16#D6
16#00,16#00,16#45,16#7D,16#45,16#00,	// 16#D7
16#00,16#00,16#45,16#7C,16#45,16#00,	// 16#D8
16#08,16#08,16#08,16#0F,16#00,16#00,	// 16#D9
16#00,16#00,16#00,16#F8,16#08,16#08,	// 16#DA
16#FF,16#FF,16#FF,16#FF,16#FF,16#FF,	// 16#DB
16#F0,16#F0,16#F0,16#F0,16#F0,16#F0,	// 16#DC
16#00,16#00,16#00,16#77,16#00,16#00,	// 16#DD
16#00,16#00,16#45,16#7D,16#44,16#00,	// 16#DE
16#0F,16#0F,16#0F,16#0F,16#0F,16#0F,	// 16#DF
16#00,16#3C,16#42,16#43,16#3D,16#00,	// 16#E0
16#00,16#FE,16#4A,16#4A,16#34,16#00,	// 16#E1
16#00,16#3C,16#43,16#43,16#3D,16#00,	// 16#E2
16#00,16#3D,16#43,16#42,16#3C,16#00,	// 16#E3
16#00,16#32,16#49,16#4A,16#31,16#00,	// 16#E4
16#00,16#3A,16#45,16#46,16#39,16#00,	// 16#E5
16#00,16#FC,16#20,16#20,16#1C,16#00,	// 16#E6
16#00,16#FE,16#AA,16#28,16#10,16#00,	// 16#E7
16#00,16#FF,16#A5,16#24,16#18,16#00,	// 16#E8
16#00,16#3C,16#40,16#41,16#3D,16#00,	// 16#E9
16#00,16#3C,16#41,16#41,16#3D,16#00,	// 16#EA
16#00,16#3D,16#41,16#40,16#3C,16#00,	// 16#EB
16#00,16#9C,16#A0,16#61,16#3D,16#00,	// 16#EC
16#00,16#04,16#08,16#71,16#09,16#04,	// 16#ED
16#00,16#00,16#02,16#02,16#02,16#00,	// 16#EE
16#00,16#00,16#07,16#03,16#00,16#00,	// 16#EF
16#00,16#00,16#08,16#08,16#08,16#00,	// 16#F0
16#00,16#00,16#24,16#2E,16#24,16#00,	// 16#F1
16#00,16#24,16#24,16#24,16#24,16#24,	// 16#F2
16#05,16#17,16#0A,16#34,16#2A,16#78,	// 16#F3
16#00,16#06,16#09,16#7F,16#01,16#7F,	// 16#F4
16#00,16#22,16#4D,16#55,16#59,16#22,	// 16#F5
16#00,16#08,16#08,16#2A,16#08,16#08,	// 16#F6
16#00,16#00,16#08,16#18,16#18,16#00,	// 16#F7
16#00,16#06,16#09,16#09,16#06,16#00,	// 16#F8
16#00,16#00,16#08,16#00,16#08,16#00,	// 16#F9
16#00,16#00,16#08,16#00,16#00,16#00,	// 16#FA
16#00,16#02,16#0F,16#00,16#00,16#00,	// 16#FB
16#00,16#09,16#0F,16#05,16#00,16#00,	// 16#FC
16#00,16#09,16#0D,16#0A,16#00,16#00,	// 16#FD
16#00,16#3C,16#3C,16#3C,16#3C,16#00,	// 16#FE
16#00,16#00,16#00,16#00,16#00,16#00 	// 16#FF
];


FONT_6X10:ARRAY[0..255,0..11]OF BYTE :=[
16#00,16#00,16#00,16#00,16#00,16#00,16#00,16#00,16#00,16#00,16#00,16#00,	// 16#00
16#70,16#00,16#D8,16#00,16#E8,16#00,16#E8,16#00,16#C8,16#00,16#70,16#00,	// 16#01
16#70,16#00,16#F8,16#00,16#B8,16#00,16#A8,16#00,16#F8,16#00,16#70,16#00,	// 16#02
16#1E,16#00,16#7E,16#00,16#FC,16#00,16#FC,16#00,16#7E,16#00,16#1E,16#00,	// 16#03
16#10,16#00,16#38,16#00,16#7C,16#00,16#FE,16#00,16#38,16#00,16#10,16#00,	// 16#04
16#38,16#00,16#38,16#00,16#FE,16#00,16#3E,16#00,16#38,16#00,16#38,16#00,	// 16#05
16#30,16#00,16#38,16#00,16#FC,16#00,16#3E,16#00,16#3C,16#00,16#30,16#00,	// 16#06
16#00,16#00,16#00,16#00,16#00,16#00,16#00,16#00,16#00,16#00,16#00,16#00,	// 16#07
16#00,16#00,16#00,16#00,16#00,16#00,16#00,16#00,16#00,16#00,16#00,16#00,	// 16#08
16#00,16#00,16#00,16#00,16#00,16#00,16#00,16#00,16#00,16#00,16#00,16#00,	// 16#09
16#00,16#00,16#00,16#00,16#00,16#00,16#00,16#00,16#00,16#00,16#00,16#00,	// 16#0A
16#70,16#00,16#88,16#00,16#88,16#00,16#8A,16#00,16#76,16#00,16#04,16#00,	// 16#0B
16#1C,16#00,16#62,16#00,16#E2,16#00,16#62,16#00,16#1C,16#00,16#00,16#00,	// 16#0C
16#00,16#00,16#00,16#00,16#00,16#00,16#00,16#00,16#00,16#00,16#00,16#00,	// 16#0D
16#80,16#01,16#80,16#01,16#FC,16#00,16#64,16#00,16#64,16#00,16#7E,16#00,	// 16#0E
16#10,16#00,16#78,16#00,16#48,16#00,16#CC,16#00,16#78,16#00,16#10,16#00,	// 16#0F
16#FC,16#00,16#78,16#00,16#78,16#00,16#38,16#00,16#10,16#00,16#10,16#00,	// 16#10
16#10,16#00,16#10,16#00,16#38,16#00,16#78,16#00,16#78,16#00,16#FC,16#00,	// 16#11
16#00,16#00,16#00,16#00,16#84,16#00,16#FE,16#01,16#84,16#00,16#00,16#00,	// 16#12
16#00,16#00,16#BE,16#00,16#00,16#00,16#BE,16#00,16#00,16#00,16#00,16#00,	// 16#13
16#06,16#00,16#0E,16#00,16#FE,16#01,16#02,16#00,16#FE,16#01,16#00,16#00,	// 16#14
16#00,16#00,16#34,16#01,16#2A,16#01,16#4A,16#01,16#B2,16#00,16#00,16#00,	// 16#15
16#18,16#00,16#18,16#00,16#18,16#00,16#18,16#00,16#18,16#00,16#18,16#00,	// 16#16
16#00,16#00,16#00,16#00,16#42,16#02,16#FF,16#02,16#42,16#02,16#00,16#00,	// 16#17
16#00,16#00,16#00,16#00,16#04,16#00,16#FE,16#01,16#04,16#00,16#00,16#00,	// 16#18
16#00,16#00,16#00,16#00,16#80,16#00,16#FE,16#01,16#80,16#00,16#00,16#00,	// 16#19
16#10,16#00,16#10,16#00,16#10,16#00,16#10,16#00,16#38,16#00,16#10,16#00,	// 16#1A
16#10,16#00,16#38,16#00,16#10,16#00,16#10,16#00,16#10,16#00,16#10,16#00,	// 16#1B
16#F8,16#00,16#80,16#00,16#80,16#00,16#80,16#00,16#80,16#00,16#80,16#00,	// 16#1C
16#10,16#00,16#38,16#00,16#10,16#00,16#10,16#00,16#38,16#00,16#10,16#00,	// 16#1D
16#80,16#00,16#E0,16#00,16#F0,16#00,16#FC,16#00,16#F0,16#00,16#80,16#00,	// 16#1E
16#04,16#00,16#1C,16#00,16#3C,16#00,16#FC,16#00,16#3C,16#00,16#04,16#00,	// 16#1F
16#00,16#00,16#00,16#00,16#00,16#00,16#00,16#00,16#00,16#00,16#00,16#00,	// 16#20
16#00,16#00,16#00,16#00,16#BE,16#00,16#00,16#00,16#00,16#00,16#00,16#00,	// 16#21
16#00,16#00,16#07,16#00,16#00,16#00,16#07,16#00,16#00,16#00,16#00,16#00,	// 16#22
16#E0,16#00,16#38,16#00,16#EE,16#00,16#38,16#00,16#2E,16#00,16#08,16#00,	// 16#23
16#8C,16#00,16#8A,16#00,16#FF,16#01,16#92,16#00,16#62,16#00,16#00,16#00,	// 16#24
16#84,16#00,16#4A,16#00,16#34,16#00,16#58,16#00,16#A4,16#00,16#42,16#00,	// 16#25
16#60,16#00,16#9C,16#00,16#BA,16#00,16#EC,16#00,16#C0,16#00,16#30,16#00,	// 16#26
16#00,16#00,16#00,16#00,16#07,16#00,16#00,16#00,16#00,16#00,16#00,16#00,	// 16#27
16#00,16#00,16#00,16#00,16#7C,16#00,16#82,16#00,16#01,16#01,16#01,16#01,	// 16#28
16#01,16#01,16#01,16#01,16#82,16#00,16#7C,16#00,16#00,16#00,16#00,16#00,	// 16#29
16#04,16#00,16#1C,16#00,16#0A,16#00,16#14,16#00,16#04,16#00,16#00,16#00,	// 16#2A
16#20,16#00,16#20,16#00,16#F8,16#00,16#20,16#00,16#20,16#00,16#00,16#00,	// 16#2B
16#00,16#00,16#00,16#00,16#C0,16#02,16#C0,16#01,16#00,16#00,16#00,16#00,	// 16#2C
16#00,16#00,16#10,16#00,16#10,16#00,16#10,16#00,16#10,16#00,16#00,16#00,	// 16#2D
16#00,16#00,16#00,16#00,16#C0,16#00,16#C0,16#00,16#00,16#00,16#00,16#00,	// 16#2E
16#00,16#01,16#C0,16#00,16#30,16#00,16#18,16#00,16#06,16#00,16#01,16#00,	// 16#2F
16#7C,16#00,16#82,16#00,16#82,16#00,16#82,16#00,16#7C,16#00,16#00,16#00,	// 16#30
16#84,16#00,16#82,16#00,16#FE,16#00,16#80,16#00,16#80,16#00,16#00,16#00,	// 16#31
16#00,16#00,16#C2,16#00,16#A2,16#00,16#92,16#00,16#8C,16#00,16#00,16#00,	// 16#32
16#00,16#00,16#82,16#00,16#92,16#00,16#92,16#00,16#6E,16#00,16#00,16#00,	// 16#33
16#30,16#00,16#28,16#00,16#24,16#00,16#FE,16#00,16#20,16#00,16#00,16#00,	// 16#34
16#00,16#00,16#9E,16#00,16#92,16#00,16#92,16#00,16#62,16#00,16#00,16#00,	// 16#35
16#78,16#00,16#A4,16#00,16#92,16#00,16#92,16#00,16#62,16#00,16#00,16#00,	// 16#36
16#00,16#00,16#C2,16#00,16#32,16#00,16#0A,16#00,16#06,16#00,16#00,16#00,	// 16#37
16#6C,16#00,16#92,16#00,16#92,16#00,16#9A,16#00,16#64,16#00,16#00,16#00,	// 16#38
16#8C,16#00,16#92,16#00,16#92,16#00,16#52,16#00,16#3C,16#00,16#00,16#00,	// 16#39
16#00,16#00,16#00,16#00,16#D8,16#00,16#D8,16#00,16#00,16#00,16#00,16#00,	// 16#3A
16#00,16#00,16#00,16#00,16#D8,16#02,16#D8,16#01,16#00,16#00,16#00,16#00,	// 16#3B
16#20,16#00,16#20,16#00,16#50,16#00,16#50,16#00,16#88,16#00,16#00,16#00,	// 16#3C
16#50,16#00,16#50,16#00,16#50,16#00,16#50,16#00,16#50,16#00,16#50,16#00,	// 16#3D
16#88,16#00,16#50,16#00,16#50,16#00,16#20,16#00,16#20,16#00,16#00,16#00,	// 16#3E
16#00,16#00,16#06,16#00,16#A2,16#00,16#12,16#00,16#0E,16#00,16#00,16#00,	// 16#3F
16#7C,16#00,16#82,16#00,16#BA,16#00,16#AA,16#00,16#BE,16#00,16#20,16#00,	// 16#40
16#80,16#00,16#78,16#00,16#26,16#00,16#2E,16#00,16#70,16#00,16#80,16#00,	// 16#41
16#FE,16#00,16#92,16#00,16#92,16#00,16#92,16#00,16#6C,16#00,16#00,16#00,	// 16#42
16#38,16#00,16#44,16#00,16#82,16#00,16#82,16#00,16#82,16#00,16#00,16#00,	// 16#43
16#FE,16#00,16#82,16#00,16#82,16#00,16#82,16#00,16#7C,16#00,16#00,16#00,	// 16#44
16#00,16#00,16#FE,16#00,16#92,16#00,16#92,16#00,16#82,16#00,16#00,16#00,	// 16#45
16#00,16#00,16#FE,16#00,16#12,16#00,16#12,16#00,16#02,16#00,16#00,16#00,	// 16#46
16#38,16#00,16#44,16#00,16#82,16#00,16#92,16#00,16#F2,16#00,16#00,16#00,	// 16#47
16#FE,16#00,16#10,16#00,16#10,16#00,16#10,16#00,16#FE,16#00,16#00,16#00,	// 16#48
16#82,16#00,16#82,16#00,16#FE,16#00,16#82,16#00,16#82,16#00,16#00,16#00,	// 16#49
16#00,16#00,16#82,16#00,16#82,16#00,16#7E,16#00,16#00,16#00,16#00,16#00,	// 16#4A
16#FE,16#00,16#10,16#00,16#28,16#00,16#44,16#00,16#82,16#00,16#00,16#00,	// 16#4B
16#00,16#00,16#FE,16#00,16#80,16#00,16#80,16#00,16#80,16#00,16#00,16#00,	// 16#4C
16#FE,16#00,16#1C,16#00,16#70,16#00,16#0C,16#00,16#FE,16#00,16#00,16#00,	// 16#4D
16#FE,16#00,16#0C,16#00,16#18,16#00,16#60,16#00,16#FE,16#00,16#00,16#00,	// 16#4E
16#7C,16#00,16#82,16#00,16#82,16#00,16#82,16#00,16#7C,16#00,16#00,16#00,	// 16#4F
16#FE,16#00,16#12,16#00,16#12,16#00,16#12,16#00,16#0C,16#00,16#00,16#00,	// 16#50
16#7C,16#00,16#82,16#00,16#82,16#00,16#82,16#00,16#7C,16#01,16#00,16#01,	// 16#51
16#FE,16#00,16#12,16#00,16#32,16#00,16#4C,16#00,16#80,16#00,16#00,16#00,	// 16#52
16#00,16#00,16#8C,16#00,16#92,16#00,16#92,16#00,16#62,16#00,16#00,16#00,	// 16#53
16#02,16#00,16#02,16#00,16#FE,16#00,16#02,16#00,16#02,16#00,16#00,16#00,	// 16#54
16#7E,16#00,16#80,16#00,16#80,16#00,16#80,16#00,16#7E,16#00,16#00,16#00,	// 16#55
16#06,16#00,16#38,16#00,16#C0,16#00,16#60,16#00,16#1C,16#00,16#02,16#00,	// 16#56
16#3E,16#00,16#E0,16#00,16#3C,16#00,16#E0,16#00,16#1E,16#00,16#00,16#00,	// 16#57
16#82,16#00,16#44,16#00,16#28,16#00,16#38,16#00,16#44,16#00,16#82,16#00,	// 16#58
16#02,16#00,16#0C,16#00,16#F0,16#00,16#0C,16#00,16#02,16#00,16#00,16#00,	// 16#59
16#C2,16#00,16#A2,16#00,16#92,16#00,16#8A,16#00,16#86,16#00,16#00,16#00,	// 16#5A
16#00,16#00,16#00,16#00,16#FF,16#01,16#01,16#01,16#01,16#01,16#00,16#00,	// 16#5B
16#01,16#00,16#06,16#00,16#18,16#00,16#20,16#00,16#C0,16#00,16#00,16#01,	// 16#5C
16#00,16#00,16#01,16#01,16#01,16#01,16#FF,16#01,16#00,16#00,16#00,16#00,	// 16#5D
16#40,16#00,16#38,16#00,16#06,16#00,16#38,16#00,16#40,16#00,16#00,16#00,	// 16#5E
16#00,16#01,16#00,16#01,16#00,16#01,16#00,16#01,16#00,16#01,16#00,16#01,	// 16#5F
16#00,16#00,16#00,16#00,16#01,16#00,16#02,16#00,16#00,16#00,16#00,16#00,	// 16#60
16#00,16#00,16#C8,16#00,16#A8,16#00,16#A8,16#00,16#F0,16#00,16#80,16#00,	// 16#61
16#FF,16#00,16#90,16#00,16#88,16#00,16#88,16#00,16#70,16#00,16#00,16#00,	// 16#62
16#70,16#00,16#88,16#00,16#88,16#00,16#88,16#00,16#88,16#00,16#00,16#00,	// 16#63
16#70,16#00,16#88,16#00,16#88,16#00,16#48,16#00,16#FF,16#00,16#00,16#00,	// 16#64
16#70,16#00,16#A8,16#00,16#A8,16#00,16#A8,16#00,16#B0,16#00,16#00,16#00,	// 16#65
16#00,16#00,16#08,16#00,16#FE,16#00,16#09,16#00,16#09,16#00,16#00,16#00,	// 16#66
16#70,16#00,16#88,16#02,16#88,16#02,16#48,16#02,16#F8,16#01,16#00,16#00,	// 16#67
16#FF,16#00,16#10,16#00,16#08,16#00,16#08,16#00,16#F8,16#00,16#00,16#00,	// 16#68
16#00,16#00,16#08,16#00,16#08,16#00,16#F9,16#00,16#00,16#00,16#00,16#00,	// 16#69
16#00,16#02,16#08,16#02,16#08,16#02,16#F9,16#01,16#00,16#00,16#00,16#00,	// 16#6A
16#00,16#00,16#FF,16#00,16#20,16#00,16#50,16#00,16#88,16#00,16#00,16#00,	// 16#6B
16#01,16#00,16#01,16#00,16#FF,16#00,16#00,16#00,16#00,16#00,16#00,16#00,	// 16#6C
16#F8,16#00,16#08,16#00,16#F8,16#00,16#08,16#00,16#F8,16#00,16#00,16#00,	// 16#6D
16#F8,16#00,16#10,16#00,16#08,16#00,16#08,16#00,16#F8,16#00,16#00,16#00,	// 16#6E
16#70,16#00,16#88,16#00,16#88,16#00,16#88,16#00,16#70,16#00,16#00,16#00,	// 16#6F
16#F8,16#03,16#90,16#00,16#88,16#00,16#88,16#00,16#70,16#00,16#00,16#00,	// 16#70
16#70,16#00,16#88,16#00,16#88,16#00,16#48,16#00,16#F8,16#03,16#00,16#00,	// 16#71
16#00,16#00,16#F8,16#00,16#10,16#00,16#08,16#00,16#18,16#00,16#00,16#00,	// 16#72
16#00,16#00,16#90,16#00,16#A8,16#00,16#A8,16#00,16#48,16#00,16#00,16#00,	// 16#73
16#00,16#00,16#08,16#00,16#7E,16#00,16#88,16#00,16#88,16#00,16#00,16#00,	// 16#74
16#F8,16#00,16#80,16#00,16#80,16#00,16#40,16#00,16#F8,16#00,16#00,16#00,	// 16#75
16#08,16#00,16#70,16#00,16#80,16#00,16#70,16#00,16#08,16#00,16#00,16#00,	// 16#76
16#38,16#00,16#C0,16#00,16#38,16#00,16#30,16#00,16#C0,16#00,16#38,16#00,	// 16#77
16#88,16#00,16#50,16#00,16#20,16#00,16#50,16#00,16#88,16#00,16#00,16#00,	// 16#78
16#08,16#02,16#30,16#02,16#C0,16#01,16#C0,16#00,16#30,16#00,16#08,16#00,	// 16#79
16#88,16#00,16#C8,16#00,16#A8,16#00,16#98,16#00,16#88,16#00,16#00,16#00,	// 16#7A
16#00,16#00,16#10,16#00,16#EF,16#01,16#01,16#01,16#01,16#01,16#00,16#00,	// 16#7B
16#00,16#00,16#00,16#00,16#FF,16#01,16#00,16#00,16#00,16#00,16#00,16#00,	// 16#7C
16#00,16#00,16#01,16#01,16#01,16#01,16#EF,16#01,16#10,16#00,16#00,16#00,	// 16#7D
16#30,16#00,16#10,16#00,16#10,16#00,16#20,16#00,16#20,16#00,16#30,16#00,	// 16#7E
16#F0,16#00,16#88,16#00,16#84,16#00,16#88,16#00,16#F0,16#00,16#00,16#00,	// 16#7F
16#38,16#00,16#44,16#00,16#82,16#02,16#82,16#03,16#82,16#00,16#00,16#00,	// 16#80
16#F8,16#00,16#82,16#00,16#80,16#00,16#42,16#00,16#F8,16#00,16#00,16#00,	// 16#81
16#70,16#00,16#A8,16#00,16#A8,16#00,16#AA,16#00,16#B1,16#00,16#00,16#00,	// 16#82
16#00,16#00,16#CA,16#00,16#A9,16#00,16#AA,16#00,16#F0,16#00,16#80,16#00,	// 16#83
16#00,16#00,16#CA,16#00,16#A8,16#00,16#AA,16#00,16#F0,16#00,16#80,16#00,	// 16#84
16#00,16#00,16#C9,16#00,16#AA,16#00,16#A8,16#00,16#F0,16#00,16#80,16#00,	// 16#85
16#00,16#00,16#C8,16#00,16#AC,16#00,16#AA,16#00,16#F4,16#00,16#80,16#00,	// 16#86
16#70,16#00,16#88,16#00,16#88,16#02,16#88,16#03,16#88,16#00,16#00,16#00,	// 16#87
16#70,16#00,16#AA,16#00,16#A9,16#00,16#AA,16#00,16#B0,16#00,16#00,16#00,	// 16#88
16#70,16#00,16#AA,16#00,16#A8,16#00,16#AA,16#00,16#B0,16#00,16#00,16#00,	// 16#89
16#70,16#00,16#A9,16#00,16#AA,16#00,16#A8,16#00,16#B0,16#00,16#00,16#00,	// 16#8A
16#00,16#00,16#0A,16#00,16#08,16#00,16#FA,16#00,16#00,16#00,16#00,16#00,	// 16#8B
16#00,16#00,16#0A,16#00,16#09,16#00,16#FA,16#00,16#00,16#00,16#00,16#00,	// 16#8C
16#00,16#00,16#09,16#00,16#0A,16#00,16#F8,16#00,16#00,16#00,16#00,16#00,	// 16#8D
16#80,16#00,16#79,16#00,16#26,16#00,16#2F,16#00,16#70,16#00,16#80,16#00,	// 16#8E
16#80,16#00,16#70,16#00,16#2D,16#00,16#27,16#00,16#39,16#00,16#C0,16#00,	// 16#8F
16#00,16#00,16#FE,16#00,16#92,16#00,16#92,16#00,16#83,16#00,16#00,16#00,	// 16#90
16#C8,16#00,16#A8,16#00,16#70,16#00,16#A8,16#00,16#A8,16#00,16#B0,16#00,	// 16#91
16#80,16#00,16#70,16#00,16#4C,16#00,16#FE,16#00,16#92,16#00,16#82,16#00,	// 16#92
16#70,16#00,16#8A,16#00,16#89,16#00,16#8A,16#00,16#70,16#00,16#00,16#00,	// 16#93
16#70,16#00,16#8A,16#00,16#88,16#00,16#8A,16#00,16#70,16#00,16#00,16#00,	// 16#94
16#70,16#00,16#89,16#00,16#8A,16#00,16#88,16#00,16#70,16#00,16#00,16#00,	// 16#95
16#F8,16#00,16#82,16#00,16#81,16#00,16#42,16#00,16#F8,16#00,16#00,16#00,	// 16#96
16#F8,16#00,16#81,16#00,16#82,16#00,16#40,16#00,16#F8,16#00,16#00,16#00,	// 16#97
16#08,16#02,16#32,16#02,16#C0,16#01,16#C2,16#00,16#30,16#00,16#08,16#00,	// 16#98
16#7C,16#00,16#83,16#00,16#82,16#00,16#83,16#00,16#7C,16#00,16#00,16#00,	// 16#99
16#7E,16#00,16#81,16#00,16#80,16#00,16#81,16#00,16#7E,16#00,16#00,16#00,	// 16#9A
16#F0,16#00,16#C8,16#00,16#A8,16#00,16#98,16#00,16#78,16#00,16#00,16#00,	// 16#9B
16#00,16#00,16#90,16#00,16#FC,16#00,16#92,16#00,16#82,16#00,16#00,16#00,	// 16#9C
16#FC,16#00,16#E2,16#00,16#9A,16#00,16#86,16#00,16#7E,16#00,16#00,16#00,	// 16#9D
16#88,16#00,16#50,16#00,16#20,16#00,16#50,16#00,16#88,16#00,16#00,16#00,	// 16#9E
16#00,16#02,16#08,16#02,16#FF,16#03,16#09,16#00,16#01,16#00,16#00,16#00,	// 16#9F
16#00,16#00,16#C8,16#00,16#A8,16#00,16#AA,16#00,16#F1,16#00,16#80,16#00,	// 16#A0
16#00,16#00,16#08,16#00,16#0A,16#00,16#F9,16#00,16#00,16#00,16#00,16#00,	// 16#A1
16#70,16#00,16#88,16#00,16#8A,16#00,16#89,16#00,16#70,16#00,16#00,16#00,	// 16#A2
16#F8,16#00,16#80,16#00,16#82,16#00,16#41,16#00,16#F8,16#00,16#00,16#00,	// 16#A3
16#F8,16#00,16#13,16#00,16#0A,16#00,16#0B,16#00,16#F8,16#00,16#00,16#00,	// 16#A4
16#FE,16#00,16#0D,16#00,16#1A,16#00,16#61,16#00,16#FE,16#00,16#00,16#00,	// 16#A5
16#00,16#00,16#1E,16#00,16#16,16#00,16#1E,16#00,16#10,16#00,16#00,16#00,	// 16#A6
16#00,16#00,16#0C,16#00,16#12,16#00,16#12,16#00,16#0C,16#00,16#00,16#00,	// 16#A7
16#00,16#00,16#80,16#03,16#40,16#02,16#28,16#02,16#00,16#03,16#00,16#00,	// 16#A8
16#1C,16#00,16#2A,16#00,16#2A,16#00,16#22,16#00,16#1C,16#00,16#00,16#00,	// 16#A9
16#10,16#00,16#10,16#00,16#10,16#00,16#10,16#00,16#70,16#00,16#00,16#00,	// 16#AA
16#82,16#00,16#6E,16#00,16#10,16#00,16#DC,16#00,16#D2,16#00,16#B0,16#00,	// 16#AB
16#82,16#00,16#6E,16#00,16#70,16#00,16#5C,16#00,16#F2,16#00,16#40,16#00,	// 16#AC
16#00,16#00,16#00,16#00,16#E8,16#03,16#00,16#00,16#00,16#00,16#00,16#00,	// 16#AD
16#20,16#00,16#50,16#00,16#A8,16#00,16#50,16#00,16#88,16#00,16#00,16#00,	// 16#AE
16#88,16#00,16#50,16#00,16#A8,16#00,16#50,16#00,16#20,16#00,16#00,16#00,	// 16#AF
16#55,16#01,16#00,16#00,16#55,16#01,16#00,16#00,16#55,16#01,16#00,16#00,	// 16#B0
16#AA,16#02,16#55,16#01,16#AA,16#02,16#55,16#01,16#AA,16#02,16#55,16#01,	// 16#B1
16#FF,16#03,16#55,16#01,16#FF,16#03,16#55,16#01,16#FF,16#03,16#55,16#01,	// 16#B2
16#00,16#00,16#00,16#00,16#00,16#00,16#FF,16#03,16#00,16#00,16#00,16#00,	// 16#B3
16#10,16#00,16#10,16#00,16#10,16#00,16#FF,16#03,16#00,16#00,16#00,16#00,	// 16#B4
16#80,16#00,16#78,16#00,16#26,16#00,16#2F,16#00,16#70,16#00,16#80,16#00,	// 16#B5
16#80,16#00,16#7A,16#00,16#27,16#00,16#2E,16#00,16#70,16#00,16#80,16#00,	// 16#B6
16#80,16#00,16#79,16#00,16#26,16#00,16#2E,16#00,16#70,16#00,16#80,16#00,	// 16#B7
16#7C,16#00,16#82,16#00,16#BA,16#00,16#AA,16#00,16#82,16#00,16#7C,16#00,	// 16#B8
16#28,16#00,16#28,16#00,16#EF,16#03,16#00,16#00,16#FF,16#03,16#00,16#00,	// 16#B9
16#00,16#00,16#00,16#00,16#FF,16#03,16#00,16#00,16#FF,16#03,16#00,16#00,	// 16#BA
16#28,16#00,16#28,16#00,16#E8,16#03,16#08,16#00,16#F8,16#03,16#00,16#00,	// 16#BB
16#28,16#00,16#28,16#00,16#2F,16#00,16#20,16#00,16#3F,16#00,16#00,16#00,	// 16#BC
16#00,16#00,16#38,16#00,16#44,16#00,16#FE,16#00,16#44,16#00,16#00,16#00,	// 16#BD
16#02,16#00,16#54,16#00,16#F8,16#00,16#58,16#00,16#04,16#00,16#02,16#00,	// 16#BE
16#10,16#00,16#10,16#00,16#10,16#00,16#F0,16#03,16#00,16#00,16#00,16#00,	// 16#BF
16#00,16#00,16#00,16#00,16#00,16#00,16#1F,16#00,16#10,16#00,16#10,16#00,	// 16#C0
16#10,16#00,16#10,16#00,16#10,16#00,16#1F,16#00,16#10,16#00,16#10,16#00,	// 16#C1
16#10,16#00,16#10,16#00,16#10,16#00,16#F0,16#03,16#10,16#00,16#10,16#00,	// 16#C2
16#00,16#00,16#00,16#00,16#00,16#00,16#FF,16#03,16#10,16#00,16#10,16#00,	// 16#C3
16#10,16#00,16#10,16#00,16#10,16#00,16#10,16#00,16#10,16#00,16#10,16#00,	// 16#C4
16#10,16#00,16#10,16#00,16#10,16#00,16#FF,16#03,16#10,16#00,16#10,16#00,	// 16#C5
16#00,16#00,16#CB,16#00,16#AA,16#00,16#AB,16#00,16#F0,16#00,16#80,16#00,	// 16#C6
16#82,16#00,16#79,16#00,16#26,16#00,16#2F,16#00,16#70,16#00,16#80,16#00,	// 16#C7
16#00,16#00,16#00,16#00,16#3F,16#00,16#20,16#00,16#2F,16#00,16#28,16#00,	// 16#C8
16#00,16#00,16#00,16#00,16#F8,16#03,16#08,16#00,16#E8,16#03,16#28,16#00,	// 16#C9
16#28,16#00,16#28,16#00,16#2F,16#00,16#20,16#00,16#2F,16#00,16#28,16#00,	// 16#CA
16#28,16#00,16#28,16#00,16#E8,16#03,16#08,16#00,16#E8,16#03,16#28,16#00,	// 16#CB
16#00,16#00,16#00,16#00,16#FF,16#03,16#00,16#00,16#EF,16#03,16#28,16#00,	// 16#CC
16#28,16#00,16#28,16#00,16#28,16#00,16#28,16#00,16#28,16#00,16#28,16#00,	// 16#CD
16#28,16#00,16#28,16#00,16#EF,16#03,16#00,16#00,16#EF,16#03,16#28,16#00,	// 16#CE
16#42,16#00,16#3C,16#00,16#24,16#00,16#24,16#00,16#3C,16#00,16#42,16#00,	// 16#CF
16#75,16#00,16#8B,16#00,16#8A,16#00,16#8D,16#00,16#78,16#00,16#00,16#00,	// 16#D0
16#FE,16#00,16#92,16#00,16#82,16#00,16#82,16#00,16#7C,16#00,16#00,16#00,	// 16#D1
16#00,16#00,16#FE,16#00,16#93,16#00,16#92,16#00,16#82,16#00,16#00,16#00,	// 16#D2
16#00,16#00,16#FF,16#00,16#92,16#00,16#93,16#00,16#82,16#00,16#00,16#00,	// 16#D3
16#00,16#00,16#FE,16#00,16#93,16#00,16#92,16#00,16#82,16#00,16#00,16#00,	// 16#D4
16#00,16#00,16#08,16#00,16#08,16#00,16#F8,16#00,16#00,16#00,16#00,16#00,	// 16#D5
16#82,16#00,16#82,16#00,16#FE,16#00,16#83,16#00,16#82,16#00,16#00,16#00,	// 16#D6
16#82,16#00,16#82,16#00,16#FF,16#00,16#82,16#00,16#82,16#00,16#00,16#00,	// 16#D7
16#82,16#00,16#83,16#00,16#FE,16#00,16#83,16#00,16#82,16#00,16#00,16#00,	// 16#D8
16#10,16#00,16#10,16#00,16#10,16#00,16#1F,16#00,16#00,16#00,16#00,16#00,	// 16#D9
16#00,16#00,16#00,16#00,16#00,16#00,16#F0,16#03,16#10,16#00,16#10,16#00,	// 16#DA
16#FF,16#03,16#FF,16#03,16#FF,16#03,16#FF,16#03,16#FF,16#03,16#FF,16#03,	// 16#DB
16#E0,16#03,16#E0,16#03,16#E0,16#03,16#E0,16#03,16#E0,16#03,16#E0,16#03,	// 16#DC
16#00,16#00,16#00,16#00,16#C7,16#01,16#00,16#00,16#00,16#00,16#00,16#00,	// 16#DD
16#82,16#00,16#82,16#00,16#FF,16#00,16#82,16#00,16#82,16#00,16#00,16#00,	// 16#DE
16#1F,16#00,16#1F,16#00,16#1F,16#00,16#1F,16#00,16#1F,16#00,16#1F,16#00,	// 16#DF
16#7C,16#00,16#82,16#00,16#82,16#00,16#83,16#00,16#7C,16#00,16#00,16#00,	// 16#E0
16#FE,16#00,16#01,16#00,16#99,16#00,16#A7,16#00,16#C0,16#00,16#00,16#00,	// 16#E1
16#7C,16#00,16#82,16#00,16#83,16#00,16#82,16#00,16#7C,16#00,16#00,16#00,	// 16#E2
16#7C,16#00,16#82,16#00,16#83,16#00,16#82,16#00,16#7C,16#00,16#00,16#00,	// 16#E3
16#70,16#00,16#8B,16#00,16#8A,16#00,16#8B,16#00,16#70,16#00,16#00,16#00,	// 16#E4
16#7E,16#00,16#83,16#00,16#82,16#00,16#83,16#00,16#7C,16#00,16#00,16#00,	// 16#E5
16#F8,16#03,16#80,16#00,16#80,16#00,16#40,16#00,16#F8,16#00,16#00,16#00,	// 16#E6
16#FF,16#03,16#90,16#00,16#88,16#00,16#88,16#00,16#70,16#00,16#00,16#00,	// 16#E7
16#FE,16#00,16#44,16#00,16#44,16#00,16#44,16#00,16#38,16#00,16#00,16#00,	// 16#E8
16#7E,16#00,16#80,16#00,16#82,16#00,16#81,16#00,16#7E,16#00,16#00,16#00,	// 16#E9
16#7E,16#00,16#82,16#00,16#81,16#00,16#82,16#00,16#7E,16#00,16#00,16#00,	// 16#EA
16#7E,16#00,16#80,16#00,16#81,16#00,16#82,16#00,16#7E,16#00,16#00,16#00,	// 16#EB
16#08,16#02,16#30,16#02,16#C0,16#01,16#C2,16#00,16#31,16#00,16#08,16#00,	// 16#EC
16#02,16#00,16#0C,16#00,16#F0,16#00,16#0E,16#00,16#03,16#00,16#00,16#00,	// 16#ED
16#01,16#00,16#01,16#00,16#01,16#00,16#01,16#00,16#01,16#00,16#01,16#00,	// 16#EE
16#00,16#00,16#00,16#00,16#02,16#00,16#01,16#00,16#00,16#00,16#00,16#00,	// 16#EF
16#00,16#00,16#10,16#00,16#10,16#00,16#10,16#00,16#10,16#00,16#00,16#00,	// 16#F0
16#90,16#00,16#90,16#00,16#FC,16#00,16#90,16#00,16#90,16#00,16#00,16#00,	// 16#F1
16#00,16#01,16#00,16#01,16#00,16#01,16#00,16#01,16#00,16#01,16#00,16#01,	// 16#F2
16#8E,16#00,16#4E,16#00,16#7A,16#00,16#58,16#00,16#F4,16#00,16#42,16#00,	// 16#F3
16#06,16#00,16#0E,16#00,16#FE,16#01,16#02,16#00,16#FE,16#01,16#00,16#00,	// 16#F4
16#00,16#00,16#34,16#01,16#2A,16#01,16#4A,16#01,16#B2,16#00,16#00,16#00,	// 16#F5
16#20,16#00,16#20,16#00,16#A8,16#00,16#20,16#00,16#20,16#00,16#00,16#00,	// 16#F6
16#00,16#00,16#00,16#00,16#00,16#02,16#00,16#03,16#00,16#00,16#00,16#00,	// 16#F7
16#00,16#00,16#04,16#00,16#0A,16#00,16#04,16#00,16#00,16#00,16#00,16#00,	// 16#F8
16#00,16#00,16#01,16#00,16#00,16#00,16#01,16#00,16#00,16#00,16#00,16#00,	// 16#F9
16#00,16#00,16#00,16#00,16#60,16#00,16#60,16#00,16#00,16#00,16#00,16#00,	// 16#FA
16#00,16#00,16#00,16#00,16#02,16#00,16#0E,16#00,16#00,16#00,16#00,16#00,	// 16#FB
16#00,16#00,16#00,16#00,16#0A,16#00,16#0E,16#00,16#0A,16#00,16#00,16#00,	// 16#FC
16#00,16#00,16#0A,16#00,16#0E,16#00,16#0A,16#00,16#00,16#00,16#00,16#00,	// 16#FD
16#F8,16#00,16#F8,16#00,16#F8,16#00,16#F8,16#00,16#F8,16#00,16#F8,16#00,	// 16#FE
16#00,16#00,16#00,16#00,16#00,16#00,16#00,16#00,16#00,16#00,16#00,16#00 	// 16#FF
];

FONT_7X12:ARRAY[0..255,0..13]OF BYTE :=[
16#00,16#00,16#00,16#00,16#00,16#00,16#00,16#00,16#00,16#00,16#00,16#00,16#00,16#00,	// 16#00
16#78,16#00,16#A4,16#00,16#4A,16#01,16#42,16#01,16#4A,16#01,16#A4,16#00,16#78,16#00,	// 16#01
16#78,16#00,16#DC,16#00,16#B6,16#01,16#BE,16#01,16#B6,16#01,16#DC,16#00,16#78,16#00,	// 16#02
16#1C,16#00,16#3E,16#00,16#7E,16#00,16#FC,16#00,16#7E,16#00,16#3E,16#00,16#1C,16#00,	// 16#03
16#10,16#00,16#38,16#00,16#7C,16#00,16#FE,16#00,16#7C,16#00,16#38,16#00,16#10,16#00,	// 16#04
16#30,16#00,16#78,16#01,16#77,16#01,16#BF,16#01,16#77,16#01,16#78,16#01,16#30,16#00,	// 16#05
16#38,16#00,16#7C,16#01,16#7E,16#01,16#BF,16#01,16#7E,16#01,16#7C,16#01,16#38,16#00,	// 16#06
16#00,16#00,16#00,16#00,16#00,16#00,16#00,16#00,16#00,16#00,16#00,16#00,16#00,16#00,	// 16#07
16#00,16#00,16#00,16#00,16#00,16#00,16#00,16#00,16#00,16#00,16#00,16#00,16#00,16#00,	// 16#08
16#00,16#00,16#00,16#00,16#00,16#00,16#00,16#00,16#00,16#00,16#00,16#00,16#00,16#00,	// 16#09
16#00,16#00,16#00,16#00,16#00,16#00,16#00,16#00,16#00,16#00,16#00,16#00,16#00,16#00,	// 16#0A
16#E0,16#00,16#10,16#01,16#10,16#01,16#1A,16#01,16#E6,16#00,16#0E,16#00,16#00,16#00,	// 16#0B
16#00,16#00,16#4E,16#00,16#51,16#00,16#F1,16#01,16#51,16#00,16#4E,16#00,16#00,16#00,	// 16#0C
16#00,16#00,16#00,16#00,16#00,16#00,16#00,16#00,16#00,16#00,16#00,16#00,16#00,16#00,	// 16#0D
16#80,16#01,16#80,16#01,16#FE,16#00,16#0A,16#00,16#C5,16#00,16#C5,16#00,16#7F,16#00,	// 16#0E
16#10,16#00,16#BA,16#00,16#44,16#00,16#C7,16#01,16#44,16#00,16#BA,16#00,16#10,16#00,	// 16#0F
16#00,16#00,16#00,16#00,16#FC,16#01,16#F8,16#00,16#70,16#00,16#20,16#00,16#00,16#00,	// 16#10
16#00,16#00,16#20,16#00,16#70,16#00,16#F8,16#00,16#FC,16#01,16#00,16#00,16#00,16#00,	// 16#11
16#00,16#00,16#44,16#00,16#C6,16#00,16#FF,16#01,16#C6,16#00,16#44,16#00,16#00,16#00,	// 16#12
16#00,16#00,16#BF,16#01,16#BF,16#01,16#00,16#00,16#BF,16#01,16#BF,16#01,16#00,16#00,	// 16#13
16#00,16#00,16#0E,16#00,16#1F,16#00,16#11,16#00,16#FF,16#01,16#01,16#00,16#FF,16#01,	// 16#14
16#00,16#00,16#8E,16#01,16#BF,16#01,16#29,16#01,16#FB,16#01,16#E3,16#00,16#00,16#00,	// 16#15
16#00,16#00,16#C0,16#01,16#C0,16#01,16#C0,16#01,16#C0,16#01,16#C0,16#01,16#00,16#00,	// 16#16
16#00,16#00,16#24,16#01,16#66,16#01,16#FF,16#01,16#66,16#01,16#24,16#01,16#00,16#00,	// 16#17
16#00,16#00,16#04,16#00,16#06,16#00,16#FF,16#01,16#06,16#00,16#04,16#00,16#00,16#00,	// 16#18
16#00,16#00,16#40,16#00,16#C0,16#00,16#FF,16#01,16#C0,16#00,16#40,16#00,16#00,16#00,	// 16#19
16#20,16#00,16#20,16#00,16#20,16#00,16#F8,16#00,16#70,16#00,16#20,16#00,16#00,16#00,	// 16#1A
16#20,16#00,16#70,16#00,16#F8,16#00,16#20,16#00,16#20,16#00,16#20,16#00,16#00,16#00,	// 16#1B
16#00,16#00,16#F0,16#01,16#00,16#01,16#00,16#01,16#00,16#01,16#00,16#01,16#00,16#00,	// 16#1C
16#20,16#00,16#70,16#00,16#F8,16#00,16#20,16#00,16#F8,16#00,16#70,16#00,16#20,16#00,	// 16#1D
16#C0,16#00,16#F0,16#00,16#FC,16#00,16#FF,16#00,16#FC,16#00,16#F0,16#00,16#C0,16#00,	// 16#1E
16#06,16#00,16#1E,16#00,16#7E,16#00,16#FE,16#01,16#7E,16#00,16#1E,16#00,16#06,16#00,	// 16#1F
16#00,16#00,16#00,16#00,16#00,16#00,16#00,16#00,16#00,16#00,16#00,16#00,16#00,16#00,	// 16#20
16#00,16#00,16#00,16#00,16#BF,16#01,16#BF,16#01,16#00,16#00,16#00,16#00,16#00,16#00,	// 16#21
16#00,16#00,16#07,16#00,16#07,16#00,16#00,16#00,16#07,16#00,16#07,16#00,16#00,16#00,	// 16#22
16#00,16#00,16#48,16#00,16#FE,16#01,16#48,16#00,16#FE,16#01,16#48,16#00,16#00,16#00,	// 16#23
16#00,16#00,16#4C,16#00,16#9E,16#00,16#93,16#03,16#F2,16#00,16#64,16#00,16#00,16#00,	// 16#24
16#00,16#00,16#C6,16#01,16#E9,16#01,16#36,16#00,16#D8,16#00,16#2F,16#01,16#C7,16#00,	// 16#25
16#00,16#00,16#E6,16#00,16#FF,16#01,16#19,16#01,16#FF,16#00,16#E6,16#01,16#30,16#01,	// 16#26
16#00,16#00,16#00,16#00,16#04,16#00,16#07,16#00,16#03,16#00,16#00,16#00,16#00,16#00,	// 16#27
16#00,16#00,16#7C,16#00,16#FE,16#00,16#83,16#01,16#01,16#01,16#00,16#00,16#00,16#00,	// 16#28
16#00,16#00,16#01,16#01,16#83,16#01,16#FE,16#00,16#7C,16#00,16#00,16#00,16#00,16#00,	// 16#29
16#10,16#00,16#54,16#00,16#7C,16#00,16#38,16#00,16#7C,16#00,16#54,16#00,16#10,16#00,	// 16#2A
16#00,16#00,16#20,16#00,16#20,16#00,16#F8,16#00,16#F8,16#00,16#20,16#00,16#20,16#00,	// 16#2B
16#00,16#00,16#00,16#00,16#80,16#05,16#80,16#07,16#80,16#03,16#00,16#00,16#00,16#00,	// 16#2C
16#00,16#00,16#20,16#00,16#20,16#00,16#20,16#00,16#20,16#00,16#20,16#00,16#00,16#00,	// 16#2D
16#00,16#00,16#00,16#00,16#80,16#01,16#80,16#01,16#80,16#01,16#00,16#00,16#00,16#00,	// 16#2E
16#00,16#01,16#C0,16#01,16#F0,16#00,16#3C,16#00,16#0F,16#00,16#03,16#00,16#00,16#00,	// 16#2F
16#00,16#00,16#FE,16#01,16#FF,16#01,16#01,16#01,16#FF,16#01,16#FF,16#00,16#00,16#00,	// 16#30
16#00,16#00,16#04,16#00,16#06,16#00,16#FF,16#01,16#FF,16#01,16#00,16#00,16#00,16#00,	// 16#31
16#00,16#00,16#86,16#01,16#C7,16#01,16#71,16#01,16#3F,16#01,16#0E,16#01,16#00,16#00,	// 16#32
16#00,16#00,16#82,16#00,16#93,16#01,16#11,16#01,16#FF,16#01,16#EE,16#00,16#00,16#00,	// 16#33
16#00,16#00,16#78,16#00,16#7F,16#00,16#47,16#00,16#F8,16#01,16#F8,16#01,16#40,16#00,	// 16#34
16#00,16#00,16#9F,16#00,16#9F,16#01,16#11,16#01,16#F1,16#01,16#E1,16#00,16#00,16#00,	// 16#35
16#00,16#00,16#F8,16#00,16#FE,16#01,16#17,16#01,16#F1,16#01,16#E0,16#00,16#00,16#00,	// 16#36
16#00,16#00,16#01,16#00,16#C1,16#01,16#F9,16#01,16#3F,16#00,16#07,16#00,16#00,16#00,	// 16#37
16#00,16#00,16#EE,16#00,16#FF,16#01,16#11,16#01,16#FF,16#01,16#EE,16#00,16#00,16#00,	// 16#38
16#00,16#00,16#0E,16#01,16#9F,16#01,16#F1,16#00,16#7F,16#00,16#1E,16#00,16#00,16#00,	// 16#39
16#00,16#00,16#00,16#00,16#8C,16#01,16#8C,16#01,16#8C,16#01,16#00,16#00,16#00,16#00,	// 16#3A
16#00,16#00,16#00,16#00,16#8C,16#05,16#8C,16#07,16#8C,16#03,16#00,16#00,16#00,16#00,	// 16#3B
16#00,16#00,16#10,16#00,16#38,16#00,16#6C,16#00,16#C6,16#00,16#83,16#01,16#00,16#00,	// 16#3C
16#00,16#00,16#48,16#00,16#48,16#00,16#48,16#00,16#48,16#00,16#48,16#00,16#00,16#00,	// 16#3D
16#00,16#00,16#83,16#01,16#C6,16#00,16#6C,16#00,16#38,16#00,16#10,16#00,16#00,16#00,	// 16#3E
16#00,16#00,16#06,16#00,16#A7,16#01,16#B1,16#01,16#1F,16#00,16#0E,16#00,16#00,16#00,	// 16#3F
16#00,16#00,16#7C,16#00,16#FE,16#00,16#83,16#01,16#39,16#01,16#45,16#01,16#3E,16#01,	// 16#40
16#00,16#00,16#FC,16#01,16#FE,16#01,16#23,16#00,16#FE,16#01,16#FC,16#01,16#00,16#00,	// 16#41
16#00,16#00,16#FF,16#01,16#FF,16#01,16#11,16#01,16#FF,16#01,16#EE,16#00,16#00,16#00,	// 16#42
16#00,16#00,16#FE,16#00,16#FF,16#01,16#01,16#01,16#C7,16#01,16#C6,16#00,16#00,16#00,	// 16#43
16#00,16#00,16#FF,16#01,16#FF,16#01,16#01,16#01,16#FF,16#01,16#FE,16#00,16#00,16#00,	// 16#44
16#00,16#00,16#FF,16#01,16#FF,16#01,16#11,16#01,16#11,16#01,16#01,16#01,16#00,16#00,	// 16#45
16#00,16#00,16#FF,16#01,16#FF,16#01,16#11,16#00,16#11,16#00,16#01,16#00,16#00,16#00,	// 16#46
16#00,16#00,16#FE,16#00,16#FF,16#01,16#01,16#01,16#F3,16#01,16#F2,16#00,16#00,16#00,	// 16#47
16#00,16#00,16#FF,16#01,16#FF,16#01,16#10,16#00,16#FF,16#01,16#FF,16#01,16#00,16#00,	// 16#48
16#00,16#00,16#00,16#00,16#01,16#01,16#FF,16#01,16#FF,16#01,16#01,16#01,16#00,16#00,	// 16#49
16#00,16#00,16#C0,16#00,16#C0,16#01,16#00,16#01,16#FF,16#01,16#FF,16#00,16#00,16#00,	// 16#4A
16#00,16#00,16#FF,16#01,16#FF,16#01,16#38,16#00,16#EF,16#01,16#C7,16#01,16#00,16#00,	// 16#4B
16#00,16#00,16#FF,16#01,16#FF,16#01,16#00,16#01,16#00,16#01,16#00,16#01,16#00,16#00,	// 16#4C
16#FF,16#01,16#FF,16#01,16#1C,16#00,16#70,16#00,16#1C,16#00,16#FF,16#01,16#FF,16#01,	// 16#4D
16#00,16#00,16#FF,16#01,16#FF,16#01,16#1C,16#00,16#30,16#00,16#FF,16#01,16#FF,16#01,	// 16#4E
16#00,16#00,16#FE,16#00,16#FF,16#01,16#01,16#01,16#FF,16#01,16#FE,16#00,16#00,16#00,	// 16#4F
16#00,16#00,16#FF,16#01,16#FF,16#01,16#11,16#00,16#1F,16#00,16#0E,16#00,16#00,16#00,	// 16#50
16#00,16#00,16#FE,16#00,16#FF,16#01,16#01,16#03,16#FF,16#07,16#FE,16#04,16#00,16#00,	// 16#51
16#00,16#00,16#FF,16#01,16#FF,16#01,16#11,16#00,16#FF,16#01,16#EE,16#01,16#00,16#00,	// 16#52
16#00,16#00,16#CE,16#00,16#9F,16#01,16#39,16#01,16#F3,16#01,16#E6,16#00,16#00,16#00,	// 16#53
16#00,16#00,16#01,16#00,16#01,16#00,16#FF,16#01,16#FF,16#01,16#01,16#00,16#01,16#00,	// 16#54
16#00,16#00,16#FF,16#00,16#FF,16#01,16#00,16#01,16#FF,16#01,16#FF,16#00,16#00,16#00,	// 16#55
16#00,16#00,16#7F,16#00,16#FF,16#00,16#80,16#01,16#FF,16#00,16#7F,16#00,16#00,16#00,	// 16#56
16#3F,16#00,16#FF,16#01,16#C0,16#01,16#3C,16#00,16#C0,16#01,16#FF,16#01,16#3F,16#00,	// 16#57
16#00,16#00,16#C7,16#01,16#EF,16#01,16#38,16#00,16#EF,16#01,16#C7,16#01,16#00,16#00,	// 16#58
16#00,16#00,16#0F,16#00,16#1F,16#00,16#F0,16#01,16#F0,16#01,16#1F,16#00,16#0F,16#00,	// 16#59
16#00,16#00,16#C1,16#01,16#F1,16#01,16#3D,16#01,16#0F,16#01,16#03,16#01,16#00,16#00,	// 16#5A
16#00,16#00,16#00,16#00,16#FF,16#07,16#FF,16#07,16#01,16#04,16#01,16#04,16#00,16#00,	// 16#5B
16#00,16#00,16#03,16#00,16#0F,16#00,16#3C,16#00,16#F0,16#00,16#C0,16#01,16#00,16#01,	// 16#5C
16#00,16#00,16#01,16#04,16#01,16#04,16#FF,16#07,16#FF,16#07,16#00,16#00,16#00,16#00,	// 16#5D
16#00,16#00,16#04,16#00,16#06,16#00,16#03,16#00,16#06,16#00,16#04,16#00,16#00,16#00,	// 16#5E
16#00,16#04,16#00,16#04,16#00,16#04,16#00,16#04,16#00,16#04,16#00,16#04,16#00,16#04,	// 16#5F
16#00,16#00,16#00,16#00,16#03,16#00,16#07,16#00,16#04,16#00,16#00,16#00,16#00,16#00,	// 16#60
16#00,16#00,16#C0,16#00,16#E8,16#01,16#28,16#01,16#F8,16#01,16#F0,16#01,16#00,16#00,	// 16#61
16#00,16#00,16#FF,16#01,16#FF,16#01,16#08,16#01,16#F8,16#01,16#F0,16#00,16#00,16#00,	// 16#62
16#00,16#00,16#F0,16#00,16#F8,16#01,16#08,16#01,16#98,16#01,16#90,16#00,16#00,16#00,	// 16#63
16#00,16#00,16#F0,16#00,16#F8,16#01,16#08,16#01,16#FF,16#01,16#FF,16#01,16#00,16#00,	// 16#64
16#00,16#00,16#F0,16#00,16#F8,16#01,16#28,16#01,16#38,16#01,16#B0,16#00,16#00,16#00,	// 16#65
16#00,16#00,16#08,16#00,16#FE,16#01,16#FF,16#01,16#09,16#00,16#09,16#00,16#00,16#00,	// 16#66
16#00,16#00,16#70,16#02,16#F8,16#04,16#88,16#04,16#F8,16#07,16#F8,16#03,16#00,16#00,	// 16#67
16#00,16#00,16#FF,16#01,16#FF,16#01,16#08,16#00,16#F8,16#01,16#F0,16#01,16#00,16#00,	// 16#68
16#00,16#00,16#00,16#00,16#08,16#01,16#F9,16#01,16#F9,16#01,16#00,16#01,16#00,16#00,	// 16#69
16#00,16#00,16#00,16#04,16#08,16#04,16#F9,16#07,16#F9,16#03,16#00,16#00,16#00,16#00,	// 16#6A
16#00,16#00,16#FF,16#01,16#FF,16#01,16#70,16#00,16#D8,16#01,16#88,16#01,16#00,16#00,	// 16#6B
16#00,16#00,16#00,16#00,16#01,16#01,16#FF,16#01,16#FF,16#01,16#00,16#01,16#00,16#00,	// 16#6C
16#F8,16#01,16#F8,16#01,16#18,16#00,16#F0,16#00,16#18,16#00,16#F8,16#01,16#F0,16#01,	// 16#6D
16#00,16#00,16#F8,16#01,16#F8,16#01,16#08,16#00,16#F8,16#01,16#F0,16#01,16#00,16#00,	// 16#6E
16#00,16#00,16#F0,16#00,16#F8,16#01,16#08,16#01,16#F8,16#01,16#F0,16#00,16#00,16#00,	// 16#6F
16#00,16#00,16#F8,16#07,16#F8,16#07,16#08,16#01,16#F8,16#01,16#F0,16#00,16#00,16#00,	// 16#70
16#00,16#00,16#F0,16#00,16#F8,16#01,16#08,16#01,16#F8,16#07,16#F8,16#07,16#00,16#00,	// 16#71
16#00,16#00,16#F8,16#01,16#F8,16#01,16#10,16#00,16#18,16#00,16#18,16#00,16#00,16#00,	// 16#72
16#00,16#00,16#30,16#01,16#78,16#01,16#68,16#01,16#E8,16#01,16#C8,16#00,16#00,16#00,	// 16#73
16#00,16#00,16#08,16#00,16#FE,16#00,16#FE,16#01,16#08,16#01,16#00,16#01,16#00,16#00,	// 16#74
16#00,16#00,16#F8,16#00,16#F8,16#01,16#00,16#01,16#F8,16#01,16#F8,16#01,16#00,16#00,	// 16#75
16#00,16#00,16#78,16#00,16#F8,16#00,16#80,16#01,16#F8,16#00,16#78,16#00,16#00,16#00,	// 16#76
16#78,16#00,16#F8,16#01,16#80,16#01,16#F0,16#00,16#80,16#01,16#F8,16#01,16#78,16#00,	// 16#77
16#00,16#00,16#98,16#01,16#F8,16#01,16#60,16#00,16#F8,16#01,16#98,16#01,16#00,16#00,	// 16#78
16#00,16#00,16#78,16#04,16#F8,16#06,16#80,16#03,16#F8,16#01,16#78,16#00,16#00,16#00,	// 16#79
16#00,16#00,16#88,16#01,16#C8,16#01,16#68,16#01,16#38,16#01,16#18,16#01,16#00,16#00,	// 16#7A
16#00,16#00,16#10,16#00,16#FE,16#00,16#EF,16#01,16#01,16#01,16#01,16#01,16#00,16#00,	// 16#7B
16#00,16#00,16#00,16#00,16#DF,16#07,16#DF,16#07,16#00,16#00,16#00,16#00,16#00,16#00,	// 16#7C
16#00,16#00,16#01,16#01,16#EF,16#01,16#FE,16#00,16#10,16#00,16#00,16#00,16#00,16#00,	// 16#7D
16#00,16#00,16#06,16#00,16#03,16#00,16#07,16#00,16#06,16#00,16#03,16#00,16#00,16#00,	// 16#7E
16#00,16#00,16#F0,16#01,16#98,16#01,16#8C,16#01,16#98,16#01,16#F0,16#01,16#00,16#00,	// 16#7F
16#00,16#00,16#FE,16#00,16#FF,16#09,16#01,16#0B,16#C7,16#05,16#C6,16#00,16#00,16#00,	// 16#80
16#00,16#00,16#FB,16#00,16#FB,16#01,16#00,16#01,16#FB,16#01,16#FB,16#01,16#00,16#00,	// 16#81
16#00,16#00,16#F0,16#00,16#FA,16#01,16#2B,16#01,16#39,16#01,16#B1,16#00,16#00,16#00,	// 16#82
16#00,16#00,16#C2,16#00,16#EB,16#01,16#29,16#01,16#FB,16#01,16#F2,16#01,16#00,16#00,	// 16#83
16#00,16#00,16#C3,16#00,16#EB,16#01,16#28,16#01,16#FB,16#01,16#F3,16#01,16#00,16#00,	// 16#84
16#00,16#00,16#C1,16#00,16#E9,16#01,16#2B,16#01,16#FA,16#01,16#F0,16#01,16#00,16#00,	// 16#85
16#00,16#00,16#C2,16#00,16#ED,16#01,16#2D,16#01,16#FA,16#01,16#F0,16#01,16#00,16#00,	// 16#86
16#00,16#00,16#F0,16#00,16#F8,16#09,16#08,16#0B,16#98,16#05,16#90,16#00,16#00,16#00,	// 16#87
16#00,16#00,16#F2,16#00,16#FB,16#01,16#29,16#01,16#3B,16#01,16#B2,16#00,16#00,16#00,	// 16#88
16#00,16#00,16#F3,16#00,16#FB,16#01,16#28,16#01,16#3B,16#01,16#B3,16#00,16#00,16#00,	// 16#89
16#00,16#00,16#F1,16#00,16#F9,16#01,16#2B,16#01,16#3A,16#01,16#B0,16#00,16#00,16#00,	// 16#8A
16#00,16#00,16#03,16#00,16#0B,16#01,16#F8,16#01,16#FB,16#01,16#03,16#01,16#00,16#00,	// 16#8B
16#00,16#00,16#0A,16#01,16#FB,16#01,16#F9,16#01,16#03,16#01,16#02,16#01,16#00,16#00,	// 16#8C
16#00,16#00,16#01,16#00,16#09,16#01,16#FB,16#01,16#FA,16#01,16#00,16#01,16#00,16#00,	// 16#8D
16#00,16#00,16#F3,16#01,16#FB,16#01,16#4C,16#00,16#FB,16#01,16#F3,16#01,16#00,16#00,	// 16#8E
16#00,16#00,16#F0,16#01,16#FA,16#01,16#4D,16#00,16#FA,16#01,16#F0,16#01,16#00,16#00,	// 16#8F
16#00,16#00,16#F8,16#01,16#FA,16#01,16#2B,16#01,16#29,16#01,16#09,16#01,16#00,16#00,	// 16#90
16#00,16#00,16#C8,16#00,16#28,16#01,16#F8,16#01,16#F8,16#00,16#48,16#01,16#70,16#01,	// 16#91
16#00,16#00,16#FE,16#01,16#23,16#00,16#FF,16#01,16#FF,16#01,16#11,16#01,16#11,16#01,	// 16#92
16#00,16#00,16#F2,16#00,16#FB,16#01,16#09,16#01,16#FB,16#01,16#F2,16#00,16#00,16#00,	// 16#93
16#00,16#00,16#F3,16#00,16#FB,16#01,16#08,16#01,16#FB,16#01,16#F3,16#00,16#00,16#00,	// 16#94
16#00,16#00,16#F1,16#00,16#F9,16#01,16#0B,16#01,16#FA,16#01,16#F0,16#00,16#00,16#00,	// 16#95
16#00,16#00,16#FA,16#00,16#FB,16#01,16#01,16#01,16#FB,16#01,16#FA,16#01,16#00,16#00,	// 16#96
16#00,16#00,16#F9,16#00,16#F9,16#01,16#03,16#01,16#FA,16#01,16#F8,16#01,16#00,16#00,	// 16#97
16#00,16#00,16#7B,16#04,16#FB,16#06,16#80,16#03,16#FB,16#01,16#7B,16#00,16#00,16#00,	// 16#98
16#00,16#00,16#F9,16#00,16#FD,16#01,16#04,16#01,16#FD,16#01,16#F9,16#00,16#00,16#00,	// 16#99
16#00,16#00,16#FD,16#00,16#FD,16#01,16#00,16#01,16#FD,16#01,16#FD,16#00,16#00,16#00,	// 16#9A
16#00,16#00,16#F0,16#03,16#F8,16#01,16#68,16#01,16#F8,16#01,16#FC,16#00,16#00,16#00,	// 16#9B
16#90,16#01,16#FE,16#01,16#7F,16#01,16#11,16#01,16#13,16#01,16#02,16#01,16#00,16#00,	// 16#9C
16#00,16#00,16#FC,16#03,16#FE,16#01,16#32,16#01,16#FE,16#01,16#FF,16#00,16#00,16#00,	// 16#9D
16#00,16#00,16#44,16#00,16#28,16#00,16#10,16#00,16#28,16#00,16#44,16#00,16#00,16#00,	// 16#9E
16#00,16#00,16#08,16#02,16#FE,16#03,16#FF,16#01,16#09,16#00,16#09,16#00,16#00,16#00,	// 16#9F
16#00,16#00,16#C0,16#00,16#EA,16#01,16#2B,16#01,16#F9,16#01,16#F1,16#01,16#00,16#00,	// 16#A0
16#00,16#00,16#00,16#00,16#0A,16#01,16#FB,16#01,16#F9,16#01,16#01,16#01,16#00,16#00,	// 16#A1
16#00,16#00,16#F0,16#00,16#FA,16#01,16#0B,16#01,16#F9,16#01,16#F1,16#00,16#00,16#00,	// 16#A2
16#00,16#00,16#F8,16#00,16#FA,16#01,16#03,16#01,16#F9,16#01,16#F9,16#01,16#00,16#00,	// 16#A3
16#00,16#00,16#FA,16#01,16#F9,16#01,16#0B,16#00,16#FA,16#01,16#F1,16#01,16#00,16#00,	// 16#A4
16#00,16#00,16#FA,16#01,16#F9,16#01,16#33,16#00,16#62,16#00,16#F9,16#01,16#F8,16#01,	// 16#A5
16#00,16#00,16#98,16#00,16#BD,16#00,16#A5,16#00,16#BF,16#00,16#BE,16#00,16#00,16#00,	// 16#A6
16#00,16#00,16#9E,16#00,16#BF,16#00,16#A1,16#00,16#BF,16#00,16#9E,16#00,16#00,16#00,	// 16#A7
16#00,16#00,16#E0,16#00,16#F0,16#01,16#1B,16#01,16#CB,16#01,16#C0,16#00,16#00,16#00,	// 16#A8
16#7C,16#00,16#82,16#00,16#7D,16#01,16#15,16#01,16#69,16#01,16#82,16#00,16#7C,16#00,	// 16#A9
16#00,16#00,16#10,16#00,16#10,16#00,16#10,16#00,16#10,16#00,16#F0,16#01,16#00,16#00,	// 16#AA
16#00,16#00,16#42,16#00,16#2F,16#00,16#10,16#00,16#98,16#01,16#D4,16#01,16#20,16#01,	// 16#AB
16#00,16#00,16#42,16#00,16#2F,16#00,16#90,16#00,16#C8,16#00,16#A4,16#00,16#F0,16#01,	// 16#AC
16#00,16#00,16#00,16#00,16#FB,16#01,16#FB,16#01,16#00,16#00,16#00,16#00,16#00,16#00,	// 16#AD
16#30,16#00,16#78,16#00,16#CC,16#00,16#B4,16#00,16#78,16#00,16#CC,16#00,16#84,16#00,	// 16#AE
16#84,16#00,16#CC,16#00,16#78,16#00,16#B4,16#00,16#CC,16#00,16#78,16#00,16#30,16#00,	// 16#AF
16#44,16#04,16#00,16#00,16#11,16#01,16#44,16#04,16#00,16#00,16#11,16#01,16#00,16#00,	// 16#B0
16#AA,16#0A,16#00,16#00,16#55,16#05,16#AA,16#0A,16#00,16#00,16#55,16#05,16#00,16#00,	// 16#B1
16#AA,16#0A,16#55,16#05,16#55,16#05,16#AA,16#0A,16#55,16#05,16#AA,16#0A,16#55,16#05,	// 16#B2
16#00,16#00,16#00,16#00,16#00,16#00,16#FF,16#0F,16#00,16#00,16#00,16#00,16#00,16#00,	// 16#B3
16#20,16#00,16#20,16#00,16#20,16#00,16#FF,16#0F,16#00,16#00,16#00,16#00,16#00,16#00,	// 16#B4
16#00,16#00,16#F0,16#01,16#FA,16#01,16#4F,16#00,16#F9,16#01,16#F1,16#01,16#00,16#00,	// 16#B5
16#00,16#00,16#F2,16#01,16#FB,16#01,16#4D,16#00,16#FB,16#01,16#F2,16#01,16#00,16#00,	// 16#B6
16#00,16#00,16#F1,16#01,16#F9,16#01,16#4F,16#00,16#FA,16#01,16#F0,16#01,16#00,16#00,	// 16#B7
16#7C,16#00,16#82,16#00,16#39,16#01,16#45,16#01,16#29,16#01,16#82,16#00,16#7C,16#00,	// 16#B8
16#50,16#00,16#50,16#00,16#DF,16#0F,16#00,16#00,16#FF,16#0F,16#00,16#00,16#00,16#00,	// 16#B9
16#00,16#00,16#00,16#00,16#FF,16#0F,16#00,16#00,16#FF,16#0F,16#00,16#00,16#00,16#00,	// 16#BA
16#50,16#00,16#50,16#00,16#D0,16#0F,16#10,16#00,16#F0,16#0F,16#00,16#00,16#00,16#00,	// 16#BB
16#50,16#00,16#50,16#00,16#5F,16#00,16#40,16#00,16#7F,16#00,16#00,16#00,16#00,16#00,	// 16#BC
16#00,16#00,16#38,16#00,16#7C,16#00,16#44,16#00,16#C7,16#01,16#44,16#00,16#00,16#00,	// 16#BD
16#00,16#00,16#A7,16#00,16#AF,16#00,16#F8,16#01,16#F8,16#01,16#AF,16#00,16#A7,16#00,	// 16#BE
16#20,16#00,16#20,16#00,16#20,16#00,16#E0,16#0F,16#00,16#00,16#00,16#00,16#00,16#00,	// 16#BF
16#00,16#00,16#00,16#00,16#00,16#00,16#3F,16#00,16#20,16#00,16#20,16#00,16#20,16#00,	// 16#C0
16#20,16#00,16#20,16#00,16#20,16#00,16#3F,16#00,16#20,16#00,16#20,16#00,16#20,16#00,	// 16#C1
16#20,16#00,16#20,16#00,16#20,16#00,16#E0,16#0F,16#20,16#00,16#20,16#00,16#20,16#00,	// 16#C2
16#00,16#00,16#00,16#00,16#00,16#00,16#FF,16#0F,16#20,16#00,16#20,16#00,16#20,16#00,	// 16#C3
16#20,16#00,16#20,16#00,16#20,16#00,16#20,16#00,16#20,16#00,16#20,16#00,16#20,16#00,	// 16#C4
16#20,16#00,16#20,16#00,16#20,16#00,16#FF,16#0F,16#20,16#00,16#20,16#00,16#20,16#00,	// 16#C5
16#00,16#00,16#C2,16#00,16#E9,16#01,16#2B,16#01,16#FA,16#01,16#F1,16#01,16#00,16#00,	// 16#C6
16#00,16#00,16#F2,16#01,16#F9,16#01,16#4F,16#00,16#FA,16#01,16#F1,16#01,16#00,16#00,	// 16#C7
16#00,16#00,16#00,16#00,16#7F,16#00,16#40,16#00,16#5F,16#00,16#50,16#00,16#50,16#00,	// 16#C8
16#00,16#00,16#00,16#00,16#F0,16#0F,16#10,16#00,16#D0,16#0F,16#50,16#00,16#50,16#00,	// 16#C9
16#50,16#00,16#50,16#00,16#5F,16#00,16#40,16#00,16#5F,16#00,16#50,16#00,16#50,16#00,	// 16#CA
16#50,16#00,16#50,16#00,16#D0,16#0F,16#10,16#00,16#D0,16#0F,16#50,16#00,16#50,16#00,	// 16#CB
16#00,16#00,16#00,16#00,16#FF,16#0F,16#00,16#00,16#DF,16#0F,16#50,16#00,16#50,16#00,	// 16#CC
16#50,16#00,16#50,16#00,16#50,16#00,16#50,16#00,16#50,16#00,16#50,16#00,16#50,16#00,	// 16#CD
16#50,16#00,16#50,16#00,16#DF,16#0F,16#00,16#00,16#DF,16#0F,16#50,16#00,16#50,16#00,	// 16#CE
16#74,16#01,16#88,16#00,16#04,16#01,16#04,16#01,16#88,16#00,16#74,16#01,16#00,16#00,	// 16#CF
16#00,16#00,16#F2,16#00,16#FF,16#01,16#0D,16#01,16#F9,16#01,16#F1,16#00,16#00,16#00,	// 16#D0
16#10,16#00,16#FF,16#01,16#FF,16#01,16#11,16#01,16#FF,16#01,16#FE,16#00,16#00,16#00,	// 16#D1
16#00,16#00,16#FA,16#01,16#FB,16#01,16#29,16#01,16#2B,16#01,16#0A,16#01,16#00,16#00,	// 16#D2
16#00,16#00,16#FB,16#01,16#FB,16#01,16#28,16#01,16#2B,16#01,16#0B,16#01,16#00,16#00,	// 16#D3
16#00,16#00,16#F9,16#01,16#F9,16#01,16#2B,16#01,16#2A,16#01,16#08,16#01,16#00,16#00,	// 16#D4
16#00,16#00,16#00,16#00,16#1E,16#00,16#1E,16#00,16#00,16#00,16#00,16#00,16#00,16#00,	// 16#D5
16#00,16#00,16#08,16#01,16#FA,16#01,16#FB,16#01,16#09,16#01,16#01,16#00,16#00,16#00,	// 16#D6
16#02,16#00,16#0B,16#01,16#F9,16#01,16#FB,16#01,16#0A,16#01,16#00,16#00,16#00,16#00,	// 16#D7
16#00,16#00,16#0B,16#01,16#FB,16#01,16#F8,16#01,16#0B,16#01,16#03,16#00,16#00,16#00,	// 16#D8
16#20,16#00,16#20,16#00,16#20,16#00,16#3F,16#00,16#00,16#00,16#00,16#00,16#00,16#00,	// 16#D9
16#00,16#00,16#00,16#00,16#00,16#00,16#E0,16#0F,16#20,16#00,16#20,16#00,16#20,16#00,	// 16#DA
16#FF,16#0F,16#FF,16#0F,16#FF,16#0F,16#FF,16#0F,16#FF,16#0F,16#FF,16#0F,16#FF,16#0F,	// 16#DB
16#C0,16#0F,16#C0,16#0F,16#C0,16#0F,16#C0,16#0F,16#C0,16#0F,16#C0,16#0F,16#C0,16#0F,	// 16#DC
16#00,16#00,16#00,16#00,16#DF,16#07,16#DF,16#07,16#00,16#00,16#00,16#00,16#00,16#00,	// 16#DD
16#01,16#00,16#09,16#01,16#FB,16#01,16#FA,16#01,16#08,16#01,16#00,16#00,16#00,16#00,	// 16#DE
16#3F,16#00,16#3F,16#00,16#3F,16#00,16#3F,16#00,16#3F,16#00,16#3F,16#00,16#3F,16#00,	// 16#DF
16#00,16#00,16#FA,16#00,16#FF,16#01,16#05,16#01,16#FD,16#01,16#F8,16#00,16#00,16#00,	// 16#E0
16#00,16#00,16#FE,16#03,16#FF,16#03,16#11,16#01,16#FF,16#01,16#EE,16#00,16#00,16#00,	// 16#E1
16#00,16#00,16#FA,16#00,16#FF,16#01,16#05,16#01,16#FF,16#01,16#FA,16#00,16#00,16#00,	// 16#E2
16#00,16#00,16#F8,16#00,16#FD,16#01,16#05,16#01,16#FF,16#01,16#FA,16#00,16#00,16#00,	// 16#E3
16#00,16#00,16#F2,16#00,16#F9,16#01,16#0B,16#01,16#FA,16#01,16#F1,16#00,16#00,16#00,	// 16#E4
16#00,16#00,16#FA,16#00,16#FD,16#01,16#07,16#01,16#FE,16#01,16#F9,16#00,16#00,16#00,	// 16#E5
16#00,16#00,16#F8,16#07,16#F8,16#07,16#00,16#01,16#F8,16#00,16#F8,16#01,16#00,16#01,	// 16#E6
16#02,16#01,16#FE,16#01,16#FE,16#01,16#4A,16#01,16#78,16#00,16#30,16#00,16#00,16#00,	// 16#E7
16#01,16#01,16#FF,16#01,16#FF,16#01,16#45,16#01,16#7C,16#00,16#38,16#00,16#00,16#00,	// 16#E8
16#00,16#00,16#F8,16#00,16#FA,16#01,16#03,16#01,16#F9,16#01,16#F9,16#00,16#00,16#00,	// 16#E9
16#00,16#00,16#FA,16#00,16#FB,16#01,16#01,16#01,16#FB,16#01,16#FA,16#00,16#00,16#00,	// 16#EA
16#00,16#00,16#F9,16#00,16#F9,16#01,16#03,16#01,16#FA,16#01,16#F8,16#00,16#00,16#00,	// 16#EB
16#00,16#00,16#78,16#04,16#FA,16#06,16#83,16#03,16#F9,16#01,16#79,16#00,16#00,16#00,	// 16#EC
16#00,16#00,16#1C,16#00,16#3E,16#00,16#E3,16#01,16#E1,16#01,16#3D,16#00,16#1C,16#00,	// 16#ED
16#00,16#00,16#00,16#00,16#04,16#00,16#04,16#00,16#04,16#00,16#04,16#00,16#00,16#00,	// 16#EE
16#00,16#00,16#00,16#00,16#02,16#00,16#03,16#00,16#01,16#00,16#01,16#00,16#00,16#00,	// 16#EF
16#00,16#00,16#00,16#00,16#20,16#00,16#20,16#00,16#20,16#00,16#20,16#00,16#00,16#00,	// 16#F0
16#00,16#00,16#10,16#01,16#10,16#01,16#7C,16#01,16#7C,16#01,16#10,16#01,16#10,16#01,	// 16#F1
16#00,16#00,16#48,16#00,16#48,16#00,16#48,16#00,16#48,16#00,16#48,16#00,16#00,16#00,	// 16#F2
16#00,16#00,16#4B,16#00,16#2F,16#00,16#95,16#00,16#C8,16#00,16#A4,16#00,16#F0,16#01,	// 16#F3
16#00,16#00,16#0E,16#00,16#1F,16#00,16#11,16#00,16#FF,16#01,16#01,16#00,16#FF,16#01,	// 16#F4
16#00,16#00,16#8E,16#01,16#BF,16#01,16#29,16#01,16#FB,16#01,16#E3,16#00,16#00,16#00,	// 16#F5
16#00,16#00,16#20,16#00,16#20,16#00,16#AC,16#01,16#AC,16#01,16#20,16#00,16#20,16#00,	// 16#F6
16#00,16#00,16#00,16#00,16#20,16#00,16#40,16#00,16#60,16#00,16#60,16#00,16#00,16#00,	// 16#F7
16#00,16#00,16#0E,16#00,16#1F,16#00,16#11,16#00,16#1F,16#00,16#0E,16#00,16#00,16#00,	// 16#F8
16#00,16#00,16#30,16#00,16#30,16#00,16#00,16#00,16#30,16#00,16#30,16#00,16#00,16#00,	// 16#F9
16#00,16#00,16#00,16#00,16#00,16#00,16#30,16#00,16#30,16#00,16#00,16#00,16#00,16#00,	// 16#FA
16#00,16#00,16#00,16#00,16#1F,16#00,16#1F,16#00,16#00,16#00,16#00,16#00,16#00,16#00,	// 16#FB
16#00,16#00,16#11,16#00,16#15,16#00,16#1F,16#00,16#0A,16#00,16#00,16#00,16#00,16#00,	// 16#FC
16#00,16#00,16#19,16#00,16#1D,16#00,16#17,16#00,16#12,16#00,16#00,16#00,16#00,16#00,	// 16#FD
16#00,16#00,16#00,16#00,16#78,16#00,16#78,16#00,16#78,16#00,16#78,16#00,16#00,16#00,	// 16#FE
16#00,16#00,16#00,16#00,16#00,16#00,16#00,16#00,16#00,16#00,16#00,16#00,16#00,16#00 	// 16#FF
];


FONT_7X12B:ARRAY[0..255,0..13]OF BYTE :=[
16#00,16#00,16#00,16#00,16#00,16#00,16#00,16#00,16#00,16#00,16#00,16#00,16#00,16#00,	// 16#00
16#F0,16#00,16#D0,16#00,16#68,16#01,16#48,16#01,16#68,16#01,16#D0,16#00,16#F0,16#00,	// 16#01
16#F0,16#00,16#F0,16#00,16#58,16#01,16#78,16#01,16#58,16#01,16#F0,16#00,16#F0,16#00,	// 16#02
16#1C,16#00,16#7E,16#00,16#FE,16#00,16#FC,16#01,16#FE,16#00,16#7E,16#00,16#1C,16#00,	// 16#03
16#10,16#00,16#38,16#00,16#7C,16#00,16#FE,16#01,16#7C,16#00,16#38,16#00,16#10,16#00,	// 16#04
16#70,16#00,16#70,16#00,16#7E,16#00,16#FE,16#01,16#FE,16#01,16#70,16#00,16#70,16#00,	// 16#05
16#70,16#00,16#78,16#00,16#7C,16#00,16#FE,16#01,16#FC,16#01,16#78,16#00,16#70,16#00,	// 16#06
16#00,16#00,16#00,16#00,16#00,16#00,16#00,16#00,16#00,16#00,16#00,16#00,16#00,16#00,	// 16#07
16#00,16#00,16#00,16#00,16#00,16#00,16#00,16#00,16#00,16#00,16#00,16#00,16#00,16#00,	// 16#08
16#00,16#00,16#00,16#00,16#00,16#00,16#00,16#00,16#00,16#00,16#00,16#00,16#00,16#00,	// 16#09
16#00,16#00,16#00,16#00,16#00,16#00,16#00,16#00,16#00,16#00,16#00,16#00,16#00,16#00,	// 16#0A
16#F0,16#00,16#08,16#01,16#08,16#01,16#08,16#01,16#0A,16#01,16#F6,16#00,16#04,16#00,	// 16#0B
16#1C,16#00,16#22,16#00,16#A2,16#00,16#E2,16#01,16#A2,16#00,16#1C,16#00,16#00,16#00,	// 16#0C
16#00,16#00,16#00,16#00,16#00,16#00,16#00,16#00,16#00,16#00,16#00,16#00,16#00,16#00,	// 16#0D
16#00,16#06,16#00,16#06,16#F8,16#03,16#8C,16#01,16#84,16#01,16#FE,16#00,16#00,16#00,	// 16#0E
16#20,16#00,16#F8,16#00,16#88,16#00,16#8C,16#01,16#88,16#00,16#F8,16#00,16#20,16#00,	// 16#0F
16#FC,16#01,16#F8,16#00,16#F8,16#00,16#70,16#00,16#70,16#00,16#20,16#00,16#20,16#00,	// 16#10
16#20,16#00,16#20,16#00,16#70,16#00,16#70,16#00,16#F8,16#00,16#F8,16#00,16#FC,16#01,	// 16#11
16#00,16#00,16#00,16#00,16#08,16#02,16#FE,16#07,16#08,16#02,16#00,16#00,16#00,16#00,	// 16#12
16#00,16#00,16#7E,16#01,16#00,16#00,16#00,16#00,16#7E,16#01,16#00,16#00,16#00,16#00,	// 16#13
16#00,16#00,16#0E,16#00,16#1E,16#00,16#FE,16#07,16#02,16#00,16#FE,16#07,16#00,16#00,	// 16#14
16#00,16#00,16#6C,16#04,16#DA,16#04,16#92,16#04,16#92,16#04,16#62,16#03,16#00,16#00,	// 16#15
16#18,16#00,16#18,16#00,16#18,16#00,16#18,16#00,16#18,16#00,16#18,16#00,16#18,16#00,	// 16#16
16#00,16#00,16#00,16#00,16#84,16#04,16#FF,16#05,16#84,16#04,16#00,16#00,16#00,16#00,	// 16#17
16#00,16#00,16#00,16#00,16#08,16#00,16#FE,16#07,16#08,16#00,16#00,16#00,16#00,16#00,	// 16#18
16#00,16#00,16#00,16#00,16#00,16#02,16#FE,16#07,16#00,16#02,16#00,16#00,16#00,16#00,	// 16#19
16#00,16#00,16#20,16#00,16#20,16#00,16#70,16#00,16#20,16#00,16#20,16#00,16#00,16#00,	// 16#1A
16#00,16#00,16#20,16#00,16#70,16#00,16#20,16#00,16#20,16#00,16#20,16#00,16#00,16#00,	// 16#1B
16#00,16#00,16#F8,16#01,16#00,16#01,16#00,16#01,16#00,16#01,16#00,16#01,16#00,16#00,	// 16#1C
16#00,16#00,16#20,16#00,16#20,16#00,16#20,16#00,16#20,16#00,16#20,16#00,16#00,16#00,	// 16#1D
16#00,16#01,16#C0,16#01,16#F0,16#01,16#FC,16#01,16#F0,16#01,16#C0,16#01,16#00,16#01,	// 16#1E
16#04,16#00,16#1C,16#00,16#7C,16#00,16#FC,16#01,16#7C,16#00,16#1C,16#00,16#04,16#00,	// 16#1F
16#00,16#00,16#00,16#00,16#00,16#00,16#00,16#00,16#00,16#00,16#00,16#00,16#00,16#00,	// 16#20
16#00,16#00,16#00,16#00,16#00,16#00,16#7E,16#01,16#00,16#00,16#00,16#00,16#00,16#00,	// 16#21
16#00,16#00,16#07,16#00,16#00,16#00,16#00,16#00,16#07,16#00,16#00,16#00,16#00,16#00,	// 16#22
16#40,16#00,16#C8,16#01,16#78,16#00,16#CE,16#01,16#78,16#00,16#4E,16#00,16#08,16#00,	// 16#23
16#00,16#00,16#0C,16#01,16#12,16#01,16#FF,16#03,16#22,16#01,16#C2,16#00,16#00,16#00,	// 16#24
16#0C,16#01,16#92,16#00,16#52,16#00,16#FC,16#00,16#28,16#01,16#24,16#01,16#C2,16#00,	// 16#25
16#E0,16#00,16#A0,16#01,16#1C,16#01,16#32,16#01,16#CA,16#01,16#8E,16#01,16#60,16#01,	// 16#26
16#00,16#00,16#00,16#00,16#00,16#00,16#07,16#00,16#00,16#00,16#00,16#00,16#00,16#00,	// 16#27
16#00,16#00,16#00,16#00,16#F8,16#00,16#06,16#03,16#03,16#06,16#01,16#04,16#00,16#00,	// 16#28
16#00,16#00,16#01,16#04,16#02,16#06,16#06,16#03,16#F8,16#00,16#00,16#00,16#00,16#00,	// 16#29
16#00,16#00,16#04,16#00,16#1C,16#00,16#0A,16#00,16#14,16#00,16#04,16#00,16#00,16#00,	// 16#2A
16#20,16#00,16#20,16#00,16#20,16#00,16#F8,16#01,16#20,16#00,16#20,16#00,16#20,16#00,	// 16#2B
16#00,16#00,16#00,16#00,16#80,16#05,16#80,16#03,16#00,16#00,16#00,16#00,16#00,16#00,	// 16#2C
16#00,16#00,16#20,16#00,16#20,16#00,16#20,16#00,16#20,16#00,16#20,16#00,16#00,16#00,	// 16#2D
16#00,16#00,16#00,16#00,16#80,16#01,16#80,16#01,16#00,16#00,16#00,16#00,16#00,16#00,	// 16#2E
16#00,16#04,16#00,16#03,16#C0,16#00,16#20,16#00,16#18,16#00,16#06,16#00,16#01,16#00,	// 16#2F
16#78,16#00,16#86,16#01,16#02,16#01,16#02,16#01,16#86,16#01,16#78,16#00,16#00,16#00,	// 16#30
16#00,16#00,16#04,16#01,16#04,16#01,16#FE,16#01,16#00,16#01,16#00,16#01,16#00,16#00,	// 16#31
16#00,16#00,16#82,16#01,16#42,16#01,16#22,16#01,16#12,16#01,16#1C,16#01,16#00,16#00,	// 16#32
16#00,16#00,16#02,16#01,16#12,16#01,16#12,16#01,16#EE,16#00,16#00,16#00,16#00,16#00,	// 16#33
16#60,16#00,16#50,16#00,16#48,16#00,16#44,16#00,16#FE,16#01,16#40,16#00,16#00,16#00,	// 16#34
16#00,16#00,16#1E,16#01,16#12,16#01,16#12,16#01,16#E2,16#00,16#00,16#00,16#00,16#00,	// 16#35
16#00,16#00,16#F8,16#00,16#24,16#01,16#12,16#01,16#12,16#01,16#E2,16#00,16#00,16#00,	// 16#36
16#00,16#00,16#82,16#01,16#62,16#00,16#12,16#00,16#0A,16#00,16#06,16#00,16#00,16#00,	// 16#37
16#00,16#00,16#EC,16#00,16#12,16#01,16#12,16#01,16#32,16#01,16#CC,16#00,16#00,16#00,	// 16#38
16#00,16#00,16#1C,16#01,16#22,16#01,16#22,16#01,16#A2,16#00,16#7C,16#00,16#00,16#00,	// 16#39
16#00,16#00,16#00,16#00,16#00,16#00,16#98,16#01,16#98,16#01,16#00,16#00,16#00,16#00,	// 16#3A
16#00,16#00,16#00,16#00,16#98,16#05,16#98,16#03,16#00,16#00,16#00,16#00,16#00,16#00,	// 16#3B
16#00,16#00,16#00,16#00,16#60,16#00,16#90,16#00,16#90,16#00,16#08,16#01,16#00,16#00,	// 16#3C
16#00,16#00,16#50,16#00,16#50,16#00,16#50,16#00,16#50,16#00,16#50,16#00,16#00,16#00,	// 16#3D
16#00,16#00,16#08,16#01,16#90,16#00,16#90,16#00,16#60,16#00,16#00,16#00,16#00,16#00,	// 16#3E
16#00,16#00,16#06,16#00,16#02,16#00,16#62,16#01,16#12,16#00,16#0C,16#00,16#00,16#00,	// 16#3F
16#78,16#00,16#84,16#00,16#72,16#01,16#4A,16#01,16#2A,16#01,16#7C,16#00,16#40,16#00,	// 16#40
16#00,16#01,16#E0,16#00,16#5C,16#00,16#42,16#00,16#5C,16#00,16#E0,16#00,16#00,16#01,	// 16#41
16#00,16#00,16#FE,16#01,16#12,16#01,16#12,16#01,16#12,16#01,16#EC,16#00,16#00,16#00,	// 16#42
16#78,16#00,16#84,16#00,16#02,16#01,16#02,16#01,16#02,16#01,16#02,16#01,16#00,16#00,	// 16#43
16#FE,16#01,16#02,16#01,16#02,16#01,16#02,16#01,16#84,16#00,16#78,16#00,16#00,16#00,	// 16#44
16#00,16#00,16#FE,16#01,16#22,16#01,16#22,16#01,16#22,16#01,16#02,16#01,16#00,16#00,	// 16#45
16#00,16#00,16#FE,16#01,16#22,16#00,16#22,16#00,16#22,16#00,16#02,16#00,16#00,16#00,	// 16#46
16#78,16#00,16#84,16#00,16#02,16#01,16#22,16#01,16#22,16#01,16#E2,16#01,16#00,16#00,	// 16#47
16#00,16#00,16#FE,16#01,16#10,16#00,16#10,16#00,16#10,16#00,16#FE,16#01,16#00,16#00,	// 16#48
16#00,16#00,16#02,16#01,16#02,16#01,16#FE,16#01,16#02,16#01,16#02,16#01,16#00,16#00,	// 16#49
16#00,16#01,16#02,16#01,16#02,16#01,16#02,16#01,16#FE,16#00,16#00,16#00,16#00,16#00,	// 16#4A
16#00,16#00,16#FE,16#01,16#30,16#00,16#48,16#00,16#84,16#00,16#02,16#01,16#00,16#00,	// 16#4B
16#00,16#00,16#FE,16#01,16#00,16#01,16#00,16#01,16#00,16#01,16#00,16#01,16#00,16#00,	// 16#4C
16#FE,16#01,16#0E,16#00,16#70,16#00,16#38,16#00,16#06,16#00,16#FE,16#01,16#00,16#00,	// 16#4D
16#00,16#00,16#FE,16#01,16#0C,16#00,16#30,16#00,16#C0,16#00,16#FE,16#01,16#00,16#00,	// 16#4E
16#78,16#00,16#86,16#01,16#02,16#01,16#02,16#01,16#86,16#01,16#78,16#00,16#00,16#00,	// 16#4F
16#00,16#00,16#FE,16#01,16#22,16#00,16#22,16#00,16#22,16#00,16#1C,16#00,16#00,16#00,	// 16#50
16#78,16#00,16#86,16#00,16#02,16#01,16#02,16#01,16#86,16#03,16#78,16#04,16#00,16#04,	// 16#51
16#00,16#00,16#FE,16#01,16#22,16#00,16#62,16#00,16#92,16#00,16#0C,16#01,16#00,16#00,	// 16#52
16#00,16#00,16#0C,16#01,16#12,16#01,16#12,16#01,16#22,16#01,16#C2,16#00,16#00,16#00,	// 16#53
16#02,16#00,16#02,16#00,16#02,16#00,16#FE,16#01,16#02,16#00,16#02,16#00,16#02,16#00,	// 16#54
16#00,16#00,16#FE,16#00,16#00,16#01,16#00,16#01,16#00,16#01,16#FE,16#00,16#00,16#00,	// 16#55
16#02,16#00,16#1C,16#00,16#E0,16#00,16#80,16#01,16#E0,16#00,16#1C,16#00,16#02,16#00,	// 16#56
16#1E,16#00,16#E0,16#01,16#E0,16#00,16#18,16#00,16#E0,16#00,16#C0,16#01,16#3E,16#00,	// 16#57
16#02,16#01,16#84,16#00,16#48,16#00,16#30,16#00,16#48,16#00,16#84,16#00,16#02,16#01,	// 16#58
16#02,16#00,16#04,16#00,16#18,16#00,16#E0,16#01,16#18,16#00,16#04,16#00,16#02,16#00,	// 16#59
16#82,16#01,16#42,16#01,16#22,16#01,16#12,16#01,16#0A,16#01,16#06,16#01,16#00,16#00,	// 16#5A
16#00,16#00,16#00,16#00,16#00,16#00,16#FF,16#07,16#01,16#04,16#01,16#04,16#01,16#04,	// 16#5B
16#01,16#00,16#06,16#00,16#18,16#00,16#20,16#00,16#C0,16#00,16#00,16#03,16#00,16#04,	// 16#5C
16#00,16#00,16#01,16#04,16#01,16#04,16#01,16#04,16#FF,16#07,16#00,16#00,16#00,16#00,	// 16#5D
16#00,16#00,16#60,16#00,16#1C,16#00,16#07,16#00,16#38,16#00,16#40,16#00,16#00,16#00,	// 16#5E
16#00,16#02,16#00,16#02,16#00,16#02,16#00,16#02,16#00,16#02,16#00,16#02,16#00,16#02,	// 16#5F
16#00,16#00,16#00,16#00,16#01,16#00,16#02,16#00,16#00,16#00,16#00,16#00,16#00,16#00,	// 16#60
16#00,16#00,16#C0,16#00,16#28,16#01,16#28,16#01,16#28,16#01,16#F0,16#01,16#00,16#01,	// 16#61
16#00,16#00,16#FF,16#01,16#10,16#01,16#08,16#01,16#08,16#01,16#F0,16#00,16#00,16#00,	// 16#62
16#00,16#00,16#F0,16#00,16#08,16#01,16#08,16#01,16#08,16#01,16#08,16#01,16#00,16#00,	// 16#63
16#00,16#00,16#F0,16#00,16#08,16#01,16#08,16#01,16#88,16#00,16#FF,16#01,16#00,16#00,	// 16#64
16#00,16#00,16#F0,16#00,16#28,16#01,16#28,16#01,16#28,16#01,16#30,16#01,16#00,16#00,	// 16#65
16#08,16#00,16#08,16#00,16#FE,16#01,16#09,16#00,16#09,16#00,16#09,16#00,16#00,16#00,	// 16#66
16#00,16#00,16#F0,16#00,16#08,16#05,16#08,16#05,16#08,16#05,16#F8,16#03,16#00,16#00,	// 16#67
16#00,16#00,16#FF,16#01,16#10,16#00,16#08,16#00,16#08,16#00,16#F8,16#01,16#00,16#00,	// 16#68
16#00,16#00,16#08,16#00,16#08,16#00,16#F9,16#01,16#00,16#00,16#00,16#00,16#00,16#00,	// 16#69
16#00,16#00,16#08,16#04,16#08,16#04,16#08,16#04,16#F9,16#03,16#00,16#00,16#00,16#00,	// 16#6A
16#00,16#00,16#FF,16#01,16#20,16#00,16#60,16#00,16#90,16#00,16#08,16#01,16#00,16#00,	// 16#6B
16#00,16#00,16#01,16#00,16#01,16#00,16#FF,16#01,16#00,16#00,16#00,16#00,16#00,16#00,	// 16#6C
16#F8,16#01,16#10,16#00,16#08,16#00,16#F8,16#01,16#10,16#00,16#08,16#00,16#F8,16#01,	// 16#6D
16#00,16#00,16#F8,16#01,16#10,16#00,16#08,16#00,16#08,16#00,16#F8,16#01,16#00,16#00,	// 16#6E
16#F0,16#00,16#08,16#01,16#08,16#01,16#08,16#01,16#08,16#01,16#F0,16#00,16#00,16#00,	// 16#6F
16#00,16#00,16#F8,16#07,16#10,16#01,16#08,16#01,16#08,16#01,16#F0,16#00,16#00,16#00,	// 16#70
16#00,16#00,16#F0,16#00,16#08,16#01,16#08,16#01,16#08,16#01,16#F8,16#07,16#00,16#00,	// 16#71
16#00,16#00,16#F8,16#01,16#10,16#00,16#08,16#00,16#08,16#00,16#18,16#00,16#00,16#00,	// 16#72
16#00,16#00,16#30,16#01,16#28,16#01,16#28,16#01,16#48,16#01,16#C8,16#00,16#00,16#00,	// 16#73
16#08,16#00,16#08,16#00,16#FE,16#00,16#08,16#01,16#08,16#01,16#08,16#01,16#00,16#00,	// 16#74
16#00,16#00,16#F8,16#01,16#00,16#01,16#00,16#01,16#80,16#00,16#F8,16#01,16#00,16#00,	// 16#75
16#08,16#00,16#30,16#00,16#C0,16#00,16#00,16#01,16#C0,16#00,16#30,16#00,16#08,16#00,	// 16#76
16#78,16#00,16#80,16#01,16#E0,16#00,16#10,16#00,16#E0,16#00,16#80,16#01,16#78,16#00,	// 16#77
16#08,16#01,16#90,16#00,16#60,16#00,16#60,16#00,16#90,16#00,16#08,16#01,16#00,16#00,	// 16#78
16#08,16#04,16#30,16#04,16#C0,16#03,16#C0,16#00,16#30,16#00,16#08,16#00,16#00,16#00,	// 16#79
16#08,16#01,16#88,16#01,16#48,16#01,16#28,16#01,16#18,16#01,16#08,16#01,16#00,16#00,	// 16#7A
16#00,16#00,16#20,16#00,16#20,16#00,16#DF,16#03,16#01,16#04,16#01,16#04,16#00,16#00,	// 16#7B
16#00,16#00,16#00,16#00,16#00,16#00,16#FF,16#07,16#00,16#00,16#00,16#00,16#00,16#00,	// 16#7C
16#00,16#00,16#01,16#04,16#01,16#04,16#DE,16#07,16#20,16#00,16#20,16#00,16#00,16#00,	// 16#7D
16#40,16#00,16#20,16#00,16#20,16#00,16#60,16#00,16#40,16#00,16#40,16#00,16#20,16#00,	// 16#7E
16#00,16#00,16#F0,16#01,16#18,16#01,16#04,16#01,16#18,16#01,16#F0,16#01,16#00,16#00,	// 16#7F
16#78,16#00,16#84,16#00,16#02,16#01,16#02,16#01,16#02,16#0B,16#02,16#0D,16#00,16#00,	// 16#80
16#00,16#00,16#F8,16#01,16#02,16#01,16#00,16#01,16#82,16#00,16#F8,16#01,16#00,16#00,	// 16#81
16#00,16#00,16#F0,16#00,16#28,16#01,16#2A,16#01,16#29,16#01,16#30,16#01,16#00,16#00,	// 16#82
16#00,16#00,16#C0,16#00,16#2A,16#01,16#29,16#01,16#29,16#01,16#F2,16#01,16#00,16#01,	// 16#83
16#00,16#00,16#C0,16#00,16#2A,16#01,16#28,16#01,16#2A,16#01,16#F0,16#01,16#00,16#01,	// 16#84
16#00,16#00,16#C0,16#00,16#29,16#01,16#2A,16#01,16#28,16#01,16#F0,16#01,16#00,16#01,	// 16#85
16#00,16#00,16#C0,16#00,16#2A,16#01,16#2D,16#01,16#2A,16#01,16#F0,16#01,16#00,16#01,	// 16#86
16#00,16#00,16#F0,16#00,16#08,16#01,16#08,16#0B,16#08,16#0D,16#08,16#01,16#00,16#00,	// 16#87
16#00,16#00,16#F0,16#00,16#2A,16#01,16#29,16#01,16#29,16#01,16#32,16#01,16#00,16#00,	// 16#88
16#00,16#00,16#F0,16#00,16#2A,16#01,16#28,16#01,16#2A,16#01,16#30,16#01,16#00,16#00,	// 16#89
16#00,16#00,16#F0,16#00,16#29,16#01,16#2A,16#01,16#28,16#01,16#30,16#01,16#00,16#00,	// 16#8A
16#00,16#00,16#08,16#00,16#0A,16#00,16#F8,16#01,16#02,16#00,16#00,16#00,16#00,16#00,	// 16#8B
16#00,16#00,16#08,16#00,16#0A,16#00,16#F9,16#01,16#01,16#00,16#02,16#00,16#00,16#00,	// 16#8C
16#00,16#00,16#08,16#00,16#09,16#00,16#FA,16#01,16#00,16#00,16#00,16#00,16#00,16#00,	// 16#8D
16#00,16#01,16#E1,16#00,16#5C,16#00,16#42,16#00,16#5D,16#00,16#E0,16#00,16#00,16#01,	// 16#8E
16#00,16#01,16#E0,16#00,16#5D,16#00,16#43,16#00,16#5D,16#00,16#E0,16#00,16#00,16#01,	// 16#8F
16#00,16#00,16#FE,16#01,16#22,16#01,16#22,16#01,16#23,16#01,16#02,16#01,16#00,16#00,	// 16#90
16#C8,16#00,16#28,16#01,16#28,16#01,16#F0,16#00,16#28,16#01,16#28,16#01,16#30,16#01,	// 16#91
16#00,16#01,16#E0,16#00,16#58,16#00,16#46,16#00,16#FE,16#01,16#22,16#01,16#02,16#01,	// 16#92
16#F0,16#00,16#08,16#01,16#0A,16#01,16#09,16#01,16#09,16#01,16#F2,16#00,16#00,16#00,	// 16#93
16#F0,16#00,16#08,16#01,16#0A,16#01,16#08,16#01,16#0A,16#01,16#F0,16#00,16#00,16#00,	// 16#94
16#F0,16#00,16#08,16#01,16#09,16#01,16#0A,16#01,16#08,16#01,16#F0,16#00,16#00,16#00,	// 16#95
16#00,16#00,16#F8,16#01,16#02,16#01,16#01,16#01,16#81,16#00,16#FA,16#01,16#00,16#00,	// 16#96
16#00,16#00,16#F9,16#01,16#02,16#01,16#00,16#01,16#80,16#00,16#F8,16#01,16#00,16#00,	// 16#97
16#08,16#04,16#30,16#04,16#C2,16#03,16#C0,16#00,16#32,16#00,16#08,16#00,16#00,16#00,	// 16#98
16#78,16#00,16#87,16#01,16#02,16#01,16#02,16#01,16#87,16#01,16#78,16#00,16#00,16#00,	// 16#99
16#00,16#00,16#FF,16#00,16#00,16#01,16#00,16#01,16#01,16#01,16#FE,16#00,16#00,16#00,	// 16#9A
16#F0,16#01,16#88,16#01,16#48,16#01,16#28,16#01,16#18,16#01,16#F8,16#00,16#00,16#00,	// 16#9B
16#00,16#00,16#00,16#00,16#90,16#01,16#7C,16#01,16#12,16#01,16#02,16#01,16#00,16#00,	// 16#9C
16#78,16#01,16#C6,16#01,16#22,16#01,16#12,16#01,16#8E,16#01,16#7A,16#00,16#00,16#00,	// 16#9D
16#08,16#01,16#90,16#00,16#60,16#00,16#60,16#00,16#90,16#00,16#08,16#01,16#00,16#00,	// 16#9E
16#00,16#04,16#00,16#04,16#08,16#04,16#FE,16#03,16#09,16#00,16#09,16#00,16#01,16#00,	// 16#9F
16#00,16#00,16#C0,16#00,16#28,16#01,16#2A,16#01,16#29,16#01,16#F0,16#01,16#00,16#01,	// 16#A0
16#00,16#00,16#08,16#00,16#08,16#00,16#FA,16#01,16#01,16#00,16#00,16#00,16#00,16#00,	// 16#A1
16#F0,16#00,16#08,16#01,16#08,16#01,16#0A,16#01,16#09,16#01,16#F0,16#00,16#00,16#00,	// 16#A2
16#00,16#00,16#F8,16#01,16#00,16#01,16#02,16#01,16#81,16#00,16#F8,16#01,16#00,16#00,	// 16#A3
16#00,16#00,16#F8,16#01,16#12,16#00,16#09,16#00,16#0A,16#00,16#F9,16#01,16#00,16#00,	// 16#A4
16#00,16#00,16#FE,16#01,16#0E,16#00,16#31,16#00,16#C2,16#00,16#FF,16#01,16#00,16#00,	// 16#A5
16#00,16#00,16#32,16#00,16#2A,16#00,16#2A,16#00,16#3E,16#00,16#20,16#00,16#00,16#00,	// 16#A6
16#00,16#00,16#1C,16#00,16#22,16#00,16#22,16#00,16#22,16#00,16#1C,16#00,16#00,16#00,	// 16#A7
16#00,16#00,16#00,16#03,16#80,16#04,16#68,16#04,16#00,16#04,16#00,16#06,16#00,16#00,	// 16#A8
16#3C,16#00,16#42,16#00,16#5A,16#00,16#5A,16#00,16#42,16#00,16#3C,16#00,16#00,16#00,	// 16#A9
16#10,16#00,16#10,16#00,16#10,16#00,16#10,16#00,16#10,16#00,16#70,16#00,16#00,16#00,	// 16#AA
16#02,16#01,16#9E,16#00,16#60,16#00,16#18,16#00,16#94,16#01,16#52,16#01,16#30,16#01,	// 16#AB
16#02,16#01,16#9E,16#00,16#60,16#00,16#D8,16#00,16#A4,16#00,16#F2,16#01,16#80,16#00,	// 16#AC
16#00,16#00,16#00,16#00,16#00,16#00,16#E8,16#07,16#00,16#00,16#00,16#00,16#00,16#00,	// 16#AD
16#00,16#00,16#20,16#00,16#50,16#00,16#A8,16#00,16#50,16#00,16#88,16#00,16#00,16#00,	// 16#AE
16#00,16#00,16#88,16#00,16#50,16#00,16#A8,16#00,16#50,16#00,16#20,16#00,16#00,16#00,	// 16#AF
16#A5,16#04,16#00,16#00,16#A5,16#04,16#00,16#00,16#00,16#00,16#A5,16#04,16#00,16#00,	// 16#B0
16#52,16#09,16#A5,16#04,16#52,16#09,16#00,16#00,16#A5,16#04,16#52,16#09,16#A5,16#04,	// 16#B1
16#FF,16#0F,16#A5,16#04,16#FF,16#0F,16#A5,16#04,16#A5,16#04,16#FF,16#0F,16#A5,16#04,	// 16#B2
16#00,16#00,16#00,16#00,16#00,16#00,16#FF,16#0F,16#00,16#00,16#00,16#00,16#00,16#00,	// 16#B3
16#20,16#00,16#20,16#00,16#20,16#00,16#FF,16#0F,16#00,16#00,16#00,16#00,16#00,16#00,	// 16#B4
16#00,16#01,16#E0,16#00,16#5E,16#00,16#43,16#00,16#5C,16#00,16#E0,16#00,16#00,16#01,	// 16#B5
16#00,16#01,16#E2,16#00,16#5D,16#00,16#43,16#00,16#5E,16#00,16#E0,16#00,16#00,16#01,	// 16#B6
16#00,16#01,16#E1,16#00,16#5E,16#00,16#42,16#00,16#5C,16#00,16#E0,16#00,16#00,16#01,	// 16#B7
16#78,16#00,16#84,16#00,16#32,16#01,16#4A,16#01,16#4A,16#01,16#84,16#00,16#78,16#00,	// 16#B8
16#50,16#00,16#50,16#00,16#DF,16#0F,16#00,16#00,16#FF,16#0F,16#00,16#00,16#00,16#00,	// 16#B9
16#00,16#00,16#00,16#00,16#FF,16#0F,16#00,16#00,16#FF,16#0F,16#00,16#00,16#00,16#00,	// 16#BA
16#50,16#00,16#50,16#00,16#D0,16#0F,16#10,16#00,16#F0,16#0F,16#00,16#00,16#00,16#00,	// 16#BB
16#50,16#00,16#50,16#00,16#5F,16#00,16#40,16#00,16#7F,16#00,16#00,16#00,16#00,16#00,	// 16#BC
16#00,16#00,16#78,16#00,16#CC,16#00,16#84,16#00,16#FE,16#01,16#84,16#00,16#00,16#00,	// 16#BD
16#02,16#00,16#A4,16#00,16#A8,16#00,16#F0,16#01,16#A8,16#00,16#A4,16#00,16#02,16#00,	// 16#BE
16#20,16#00,16#20,16#00,16#20,16#00,16#E0,16#0F,16#00,16#00,16#00,16#00,16#00,16#00,	// 16#BF
16#00,16#00,16#00,16#00,16#00,16#00,16#3F,16#00,16#20,16#00,16#20,16#00,16#20,16#00,	// 16#C0
16#20,16#00,16#20,16#00,16#20,16#00,16#3F,16#00,16#20,16#00,16#20,16#00,16#20,16#00,	// 16#C1
16#20,16#00,16#20,16#00,16#20,16#00,16#E0,16#0F,16#20,16#00,16#20,16#00,16#20,16#00,	// 16#C2
16#00,16#00,16#00,16#00,16#00,16#00,16#FF,16#0F,16#20,16#00,16#20,16#00,16#20,16#00,	// 16#C3
16#20,16#00,16#20,16#00,16#20,16#00,16#20,16#00,16#20,16#00,16#20,16#00,16#20,16#00,	// 16#C4
16#20,16#00,16#20,16#00,16#20,16#00,16#FF,16#0F,16#20,16#00,16#20,16#00,16#20,16#00,	// 16#C5
16#00,16#00,16#C0,16#00,16#2A,16#01,16#29,16#01,16#2A,16#01,16#F1,16#01,16#00,16#01,	// 16#C6
16#00,16#01,16#E0,16#00,16#5E,16#00,16#43,16#00,16#5E,16#00,16#E1,16#00,16#00,16#01,	// 16#C7
16#00,16#00,16#00,16#00,16#7F,16#00,16#40,16#00,16#5F,16#00,16#50,16#00,16#50,16#00,	// 16#C8
16#00,16#00,16#00,16#00,16#F0,16#0F,16#10,16#00,16#D0,16#0F,16#50,16#00,16#50,16#00,	// 16#C9
16#50,16#00,16#50,16#00,16#5F,16#00,16#40,16#00,16#5F,16#00,16#50,16#00,16#50,16#00,	// 16#CA
16#50,16#00,16#50,16#00,16#D0,16#0F,16#10,16#00,16#D0,16#0F,16#50,16#00,16#50,16#00,	// 16#CB
16#00,16#00,16#00,16#00,16#FF,16#0F,16#00,16#00,16#DF,16#0F,16#50,16#00,16#50,16#00,	// 16#CC
16#50,16#00,16#50,16#00,16#50,16#00,16#50,16#00,16#50,16#00,16#50,16#00,16#50,16#00,	// 16#CD
16#50,16#00,16#50,16#00,16#DF,16#0F,16#00,16#00,16#DF,16#0F,16#50,16#00,16#50,16#00,	// 16#CE
16#82,16#00,16#7C,16#00,16#44,16#00,16#44,16#00,16#44,16#00,16#7C,16#00,16#82,16#00,	// 16#CF
16#F1,16#00,16#0D,16#01,16#0A,16#01,16#0F,16#01,16#0C,16#01,16#F8,16#00,16#00,16#00,	// 16#D0
16#FE,16#01,16#12,16#01,16#02,16#01,16#02,16#01,16#84,16#00,16#78,16#00,16#00,16#00,	// 16#D1
16#00,16#00,16#FE,16#01,16#23,16#01,16#23,16#01,16#22,16#01,16#02,16#01,16#00,16#00,	// 16#D2
16#00,16#00,16#FF,16#01,16#22,16#01,16#22,16#01,16#23,16#01,16#02,16#01,16#00,16#00,	// 16#D3
16#00,16#00,16#FE,16#01,16#23,16#01,16#22,16#01,16#22,16#01,16#02,16#01,16#00,16#00,	// 16#D4
16#00,16#00,16#08,16#00,16#08,16#00,16#F8,16#01,16#00,16#00,16#00,16#00,16#00,16#00,	// 16#D5
16#00,16#00,16#02,16#01,16#02,16#01,16#FE,16#01,16#03,16#01,16#02,16#01,16#00,16#00,	// 16#D6
16#00,16#00,16#02,16#01,16#03,16#01,16#FF,16#01,16#02,16#01,16#02,16#01,16#00,16#00,	// 16#D7
16#00,16#00,16#03,16#01,16#02,16#01,16#FE,16#01,16#03,16#01,16#02,16#01,16#00,16#00,	// 16#D8
16#20,16#00,16#20,16#00,16#20,16#00,16#3F,16#00,16#00,16#00,16#00,16#00,16#00,16#00,	// 16#D9
16#00,16#00,16#00,16#00,16#00,16#00,16#E0,16#0F,16#20,16#00,16#20,16#00,16#20,16#00,	// 16#DA
16#FF,16#0F,16#FF,16#0F,16#FF,16#0F,16#FF,16#0F,16#FF,16#0F,16#FF,16#0F,16#FF,16#0F,	// 16#DB
16#C0,16#0F,16#C0,16#0F,16#C0,16#0F,16#C0,16#0F,16#C0,16#0F,16#C0,16#0F,16#C0,16#0F,	// 16#DC
16#00,16#00,16#00,16#00,16#00,16#00,16#8F,16#07,16#00,16#00,16#00,16#00,16#00,16#00,	// 16#DD
16#00,16#00,16#02,16#01,16#03,16#01,16#FE,16#01,16#02,16#01,16#02,16#01,16#00,16#00,	// 16#DE
16#3F,16#00,16#3F,16#00,16#3F,16#00,16#3F,16#00,16#3F,16#00,16#3F,16#00,16#3F,16#00,	// 16#DF
16#78,16#00,16#86,16#01,16#02,16#01,16#02,16#01,16#87,16#01,16#78,16#00,16#00,16#00,	// 16#E0
16#00,16#00,16#FF,16#01,16#01,16#00,16#19,16#01,16#27,16#01,16#40,16#01,16#80,16#00,	// 16#E1
16#78,16#00,16#86,16#01,16#03,16#01,16#03,16#01,16#86,16#01,16#78,16#00,16#00,16#00,	// 16#E2
16#78,16#00,16#86,16#01,16#03,16#01,16#02,16#01,16#86,16#01,16#78,16#00,16#00,16#00,	// 16#E3
16#F0,16#00,16#08,16#01,16#0A,16#01,16#09,16#01,16#0A,16#01,16#F1,16#00,16#00,16#00,	// 16#E4
16#78,16#00,16#86,16#01,16#02,16#01,16#03,16#01,16#86,16#01,16#79,16#00,16#00,16#00,	// 16#E5
16#00,16#00,16#F8,16#07,16#00,16#01,16#00,16#01,16#80,16#00,16#F8,16#01,16#00,16#00,	// 16#E6
16#00,16#00,16#FF,16#07,16#10,16#01,16#08,16#01,16#08,16#01,16#F0,16#00,16#00,16#00,	// 16#E7
16#00,16#00,16#FE,16#01,16#84,16#00,16#84,16#00,16#84,16#00,16#78,16#00,16#00,16#00,	// 16#E8
16#00,16#00,16#FE,16#00,16#00,16#01,16#02,16#01,16#01,16#01,16#FE,16#00,16#00,16#00,	// 16#E9
16#00,16#00,16#FE,16#00,16#01,16#01,16#01,16#01,16#02,16#01,16#FE,16#00,16#00,16#00,	// 16#EA
16#00,16#00,16#FE,16#00,16#01,16#01,16#02,16#01,16#00,16#01,16#FE,16#00,16#00,16#00,	// 16#EB
16#08,16#04,16#30,16#04,16#C0,16#03,16#C2,16#00,16#31,16#00,16#08,16#00,16#00,16#00,	// 16#EC
16#02,16#00,16#04,16#00,16#18,16#00,16#E2,16#01,16#19,16#00,16#04,16#00,16#02,16#00,	// 16#ED
16#01,16#00,16#01,16#00,16#01,16#00,16#01,16#00,16#01,16#00,16#01,16#00,16#01,16#00,	// 16#EE
16#00,16#00,16#00,16#00,16#02,16#00,16#01,16#00,16#00,16#00,16#00,16#00,16#00,16#00,	// 16#EF
16#00,16#00,16#20,16#00,16#20,16#00,16#20,16#00,16#20,16#00,16#20,16#00,16#00,16#00,	// 16#F0
16#00,16#00,16#10,16#01,16#10,16#01,16#7C,16#01,16#10,16#01,16#10,16#01,16#00,16#00,	// 16#F1
16#00,16#0A,16#00,16#0A,16#00,16#0A,16#00,16#0A,16#00,16#0A,16#00,16#0A,16#00,16#0A,	// 16#F2
16#16,16#01,16#96,16#00,16#5E,16#00,16#F0,16#00,16#A8,16#00,16#F4,16#01,16#82,16#00,	// 16#F3
16#00,16#00,16#0E,16#00,16#1E,16#00,16#FE,16#07,16#02,16#00,16#FE,16#07,16#00,16#00,	// 16#F4
16#00,16#00,16#6C,16#04,16#DA,16#04,16#92,16#04,16#92,16#04,16#62,16#03,16#00,16#00,	// 16#F5
16#20,16#00,16#20,16#00,16#28,16#01,16#20,16#00,16#20,16#00,16#20,16#00,16#00,16#00,	// 16#F6
16#00,16#00,16#00,16#00,16#00,16#00,16#00,16#0A,16#00,16#0C,16#00,16#00,16#00,16#00,	// 16#F7
16#00,16#00,16#00,16#00,16#04,16#00,16#0A,16#00,16#04,16#00,16#00,16#00,16#00,16#00,	// 16#F8
16#00,16#00,16#01,16#00,16#00,16#00,16#00,16#00,16#01,16#00,16#00,16#00,16#00,16#00,	// 16#F9
16#00,16#00,16#00,16#00,16#60,16#00,16#60,16#00,16#00,16#00,16#00,16#00,16#00,16#00,	// 16#FA
16#00,16#00,16#00,16#00,16#02,16#00,16#1E,16#00,16#00,16#00,16#00,16#00,16#00,16#00,	// 16#FB
16#00,16#00,16#00,16#00,16#12,16#00,16#16,16#00,16#16,16#00,16#1E,16#00,16#00,16#00,	// 16#FC
16#00,16#00,16#00,16#00,16#12,16#00,16#1A,16#00,16#1A,16#00,16#16,16#00,16#00,16#00,	// 16#FD
16#F8,16#01,16#F8,16#01,16#F8,16#01,16#F8,16#01,16#F8,16#01,16#F8,16#01,16#F8,16#01,	// 16#FE
16#00,16#00,16#00,16#00,16#00,16#00,16#00,16#00,16#00,16#00,16#00,16#00,16#00,16#00 	// 16#FF
];


